METHOD TryMakeReferenceTo : BOOL
VAR_INPUT
	Target : I_Datatype;
END_VAR
VAR
	targetAsBit : I_BIT;
END_VAR
IF NOT Target.Root.TryResolveAs_BIT(targetAsBit) THEN
	RETURN;
END_IF

MakeReferenceTo(targetAsBit.Parent, targetAsBit.ByteOffset, targetAsBit.BitOffset);
TryMakeReferenceTo := TRUE;
END_METHOD

METHOD PUBLIC TryResolveAs_BIT : BOOL
VAR_INPUT
	Destination : REFERENCE TO I_BIT;
END_VAR
Destination := THIS^;
TryResolveAs_BIT := TRUE;
END_METHOD

PROPERTY PUBLIC TypeName : T_MAXSTRING
GET
TypeName := 'BIT';
END_GET
END_PROPERTY

PROPERTY PUBLIC Value : BOOL
GET
Value := GetBitValue();
END_GET
SET
SetBitValue(Value);
END_SET
END_PROPERTY

END_FUNCTION_BLOCK

// mobject-datatypes/Primitive/_NULL
{attribute 'linkalways'} 
{attribute 'no_explicit_call' := 'This FB is a CLASS and must be accessed using methods or properties'}
{attribute 'enable_dynamic_creation'}
FUNCTION_BLOCK _NULL EXTENDS DatatypeBase
VAR
END_VAR

PROPERTY PUBLIC Address : PVOID
GET
Address := 0;
END_GET
END_PROPERTY

METHOD PUBLIC ClearReference
VAR_INPUT
END_VAR
END_METHOD

METHOD PUBLIC Clone : I_Datatype
VAR
    pClone : POINTER TO _NULL;
END_VAR
pClone := __NEW(_NULL);
Clone := pClone^;
END_METHOD

PROPERTY PUBLIC IsNull : BOOL
GET
IsNull := TRUE;
END_GET
END_PROPERTY

METHOD PUBLIC SerializeWith
VAR_INPUT
	Serializer : I_Serializer;
END_VAR
Serializer.AddNull();
END_METHOD

PROPERTY PUBLIC Size : UDINT
GET
Size := 0;
END_GET
END_PROPERTY

METHOD TryDeserializeFrom : BOOL
VAR_INPUT
	Deserializer : I_Deserializer;
	Feedback : I_DeserializerFeedback;
END_VAR
END_METHOD

METHOD TryMakeReferenceTo : BOOL
VAR_INPUT
	Target : I_Datatype;
END_VAR
TryMakeReferenceTo := FALSE;
END_METHOD

PROPERTY PUBLIC TypeName : T_MAXSTRING
GET
TypeName := 'NULL';
END_GET
END_PROPERTY

END_FUNCTION_BLOCK

// mobject-datatypes/Primitive/_PVOID
{attribute 'linkalways'} 
{attribute 'no_explicit_call' := 'This FB is a CLASS and must be accessed using methods or properties'}
{attribute 'enable_dynamic_creation'}
FUNCTION_BLOCK _PVOID EXTENDS DatatypeBase IMPLEMENTS I_PVOID
VAR
	localData : PVOID;
	activeData : REFERENCE TO PVOID REF= localData;
END_VAR

PROPERTY PUBLIC Address : PVOID
GET
Address := ADR(activeData);
END_GET
END_PROPERTY

METHOD PUBLIC ClearReference
VAR_INPUT
END_VAR
activeData REF= localData;
END_METHOD

METHOD PUBLIC Clone : I_Datatype
VAR
    pClone : POINTER TO _PVOID;
END_VAR
pClone := __NEW(_PVOID);
Clone := pClone^;
END_METHOD

METHOD PUBLIC MakeReferenceTo
VAR_INPUT
	ReferenceTarget : REFERENCE TO PVOID;
END_VAR
activeData REF= ReferenceTarget;
END_METHOD

METHOD PUBLIC SerializeWith
VAR_INPUT
	Serializer : I_Serializer;
END_VAR
VAR
	pVoidAsString : T_MAXSTRING;
END_VAR
pVoidAsString := pvoid_To_string(activeData);
Serializer.AddString(pVoidAsString);
END_METHOD

PROPERTY PUBLIC Size : UDINT
GET
Size := SIZEOF(activeData);
END_GET
END_PROPERTY

METHOD TryDeserializeFrom : BOOL
VAR_INPUT
	Deserializer : I_Deserializer;
	Feedback : I_DeserializerFeedback;
END_VAR
VAR
	pVoidAsString : T_MAXSTRING;
END_VAR
IF NOT Deserializer.TryGetString(pVoidAsString, Feedback) THEN
	RETURN;
END_IF

activeData := STRING_TO_PVOID(pVoidAsString);
TryDeserializeFrom := TRUE;
END_METHOD

METHOD TryMakeReferenceTo : BOOL
VAR_INPUT
	Target : I_Datatype;
END_VAR
VAR
	pTargetData : POINTER TO PVOID;
END_VAR
IF NOT IsEquivalentTo(Target) THEN
	RETURN;
END_IF

pTargetData := Target.Address;
activeData REF= pTargetData^;
TryMakeReferenceTo := TRUE;
END_METHOD

METHOD PUBLIC TryResolveAs_PVOID : BOOL
VAR_INPUT
	Destination : REFERENCE TO I_PVOID;
END_VAR
Destination := THIS^;
TryResolveAs_PVOID := TRUE;
END_METHOD

PROPERTY PUBLIC TypeName : T_MAXSTRING
GET
TypeName := 'PVOID';
END_GET
END_PROPERTY

{warning disable C5410}
PROPERTY PUBLIC Value : REFERENCE TO PVOID
{warning restore C5410}
GET
Value REF= activeData;
END_GET
END_PROPERTY

END_FUNCTION_BLOCK

// mobject-datatypes/Primitive/_REFERENCE_TO
{attribute 'linkalways'} 
{attribute 'no_explicit_call' := 'This FB is a CLASS and must be accessed using methods or properties'}
{attribute 'enable_dynamic_creation'}
FUNCTION_BLOCK _REFERENCE_TO EXTENDS Disposable IMPLEMENTS I_REFERENCE_TO
VAR
	nullTarget : _NULL;
	_target : I_Datatype := nullTarget;
END_VAR

//FB_Init is always available implicitly and it is used primarily for initialization.
//The return value is not evaluated. For a specific influence, you can also declare the
//methods explicitly and provide additional code there with the standard initialization
//code. You can evaluate the return value.
METHOD FB_Init: BOOL
VAR_INPUT
    bInitRetains: BOOL; // TRUE: the retain variables are initialized (reset warm / reset cold)
    bInCopyCode: BOOL;  // TRUE: the instance will be copied to the copy code afterward (online change)  
	RefTo : I_Datatype; 
END_VAR
IF RefTo = 0 THEN
	RETURN;
END_IF

this^._target := RefTo;
END_METHOD

METHOD PUBLIC Accept
VAR_INPUT
	Visitor : I_DatatypeVisitor;
END_VAR
Visitor.VisitDatatype(THIS^);
END_METHOD

PROPERTY PUBLIC Address : PVOID
GET
Address := _target.Address;
END_GET
END_PROPERTY

METHOD PUBLIC ClearReference
VAR_INPUT
END_VAR
_target := nullTarget;
END_METHOD

METHOD PUBLIC Clone : I_Datatype
VAR
    pClone : POINTER TO _REFERENCE_TO;
END_VAR
pClone := __NEW(_REFERENCE_TO(RefTo := _target));
Clone := pClone^;
END_METHOD

METHOD PUBLIC IsEquivalentTo : BOOL
VAR_INPUT
	Datatype : I_Datatype;
END_VAR
IsEquivalentTo := _target.IsEquivalentTo(Datatype);
END_METHOD

PROPERTY PUBLIC IsNull : BOOL
GET
IsNull := _target.IsNull;
END_GET
END_PROPERTY

PROPERTY PUBLIC IsUserDefined : BOOL
GET
IsUserDefined := _target.IsUserDefined;
END_GET
END_PROPERTY

PROPERTY PUBLIC IsValidReference : BOOL
GET
IF _target.IsNull THEN
	RETURN;
END_IF

IsValidReference := TRUE;
END_GET
END_PROPERTY

PROPERTY PUBLIC Root : I_Datatype
GET
IF _target.IsNull THEN
	Root := THIS^;
	RETURN;
END_IF

Root := _target.Root;
END_GET
END_PROPERTY

METHOD PUBLIC SerializeTypeWith
VAR_INPUT
	Serializer : I_Serializer;
END_VAR
Serializer.StartObject();
Serializer.AddKeyString('typeName',TypeName);
Serializer.EndObject();
END_METHOD

METHOD PUBLIC SerializeWith
VAR_INPUT
	Serializer : I_Serializer;
END_VAR
_target.SerializeWith(Serializer);
END_METHOD

PROPERTY PUBLIC Size : UDINT
GET
Size := _target.Size;
END_GET
END_PROPERTY

METHOD PUBLIC TryConvertTo : BOOL
VAR_INPUT
	Destination : ANY;
END_VAR
TryConvertTo := _target.TryConvertTo(Destination);
END_METHOD

METHOD PUBLIC TryConvertTo_ : BOOL
VAR_INPUT
	Destination : I_Datatype;
END_VAR
TryConvertTo_ := _target.TryConvertTo_(Destination);
END_METHOD

METHOD PUBLIC TryCopyFrom : BOOL
VAR_INPUT
	Source : I_Datatype;
END_VAR
TryCopyFrom := _target.TryCopyFrom(Source);
END_METHOD

METHOD TryDeserializeFrom : BOOL
VAR_INPUT
	Deserializer : I_Deserializer;
	Feedback : I_DeserializerFeedback;
END_VAR
TryDeserializeFrom := _target.TryDeserializeFrom(Deserializer, Feedback);
END_METHOD

METHOD TryMakeReferenceTo : BOOL
VAR_INPUT
	Target : I_Datatype;
END_VAR
IF Target = 0 THEN
	RETURN;
END_IF

_target := Target;
TryMakeReferenceTo := TRUE;
END_METHOD

METHOD PUBLIC TryResolveAs_ANY : BOOL
VAR_INPUT
	Destination : REFERENCE TO I_ANY;
END_VAR
TryResolveAs_ANY := _target.TryResolveAs_ANY(Destination);
END_METHOD

METHOD PUBLIC TryResolveAs_BIT : BOOL
VAR_INPUT
	Destination : REFERENCE TO I_BIT;
END_VAR
TryResolveAs_BIT := _target.TryResolveAs_BIT(Destination);
END_METHOD

METHOD PUBLIC TryResolveAs_BOOL : BOOL
VAR_INPUT
	Destination : REFERENCE TO I_BOOL;
END_VAR
TryResolveAs_BOOL := _target.TryResolveAs_BOOL(Destination);
END_METHOD

METHOD PUBLIC TryResolveAs_BYTE : BOOL
VAR_INPUT
	Destination : REFERENCE TO I_BYTE;
END_VAR
TryResolveAs_BYTE := _target.TryResolveAs_BYTE(Destination);
END_METHOD

METHOD PUBLIC TryResolveAs_DINT : BOOL
VAR_INPUT
	Destination : REFERENCE TO I_DINT;
END_VAR
TryResolveAs_DINT := _target.TryResolveAs_DINT(Destination);
END_METHOD

METHOD PUBLIC TryResolveAs_DT : BOOL
VAR_INPUT
	Destination : REFERENCE TO I_DT;
END_VAR
TryResolveAs_DT := _target.TryResolveAs_DT(Destination);
END_METHOD

METHOD PUBLIC TryResolveAs_DWORD : BOOL
VAR_INPUT
	Destination : REFERENCE TO I_DWORD;
END_VAR
TryResolveAs_DWORD := _target.TryResolveAs_DWORD(Destination);
END_METHOD

METHOD PUBLIC TryResolveAs_INT : BOOL
VAR_INPUT
	Destination : REFERENCE TO I_INT;
END_VAR
TryResolveAs_INT := _target.TryResolveAs_INT(Destination);
END_METHOD

METHOD PUBLIC TryResolveAs_LINT : BOOL
VAR_INPUT
	Destination : REFERENCE TO I_LINT;
END_VAR
TryResolveAs_LINT := _target.TryResolveAs_LINT(Destination);
END_METHOD

METHOD PUBLIC TryResolveAs_LREAL : BOOL
VAR_INPUT
	Destination : REFERENCE TO I_LREAL;
END_VAR
TryResolveAs_LREAL := _target.TryResolveAs_LREAL(Destination);
END_METHOD

METHOD PUBLIC TryResolveAs_LWORD : BOOL
VAR_INPUT
	Destination : REFERENCE TO I_LWORD;
END_VAR
TryResolveAs_LWORD := _target.TryResolveAs_LWORD(Destination);
END_METHOD

METHOD PUBLIC TryResolveAs_PVOID : BOOL
VAR_INPUT
	Destination : REFERENCE TO I_PVOID;
END_VAR
TryResolveAs_PVOID := _target.TryResolveAs_PVOID(Destination);
END_METHOD

METHOD PUBLIC TryResolveAs_REAL : BOOL
VAR_INPUT
	Destination : REFERENCE TO I_REAL;
END_VAR
TryResolveAs_REAL := _target.TryResolveAs_REAL(Destination);
END_METHOD

METHOD PUBLIC TryResolveAs_REFERENCE_TO : BOOL
VAR_INPUT
	Destination : REFERENCE TO I_REFERENCE_TO;
END_VAR
Destination := THIS^;
TryResolveAs_REFERENCE_TO := TRUE;
END_METHOD

METHOD PUBLIC TryResolveAs_SINT : BOOL
VAR_INPUT
	Destination : REFERENCE TO I_SINT;
END_VAR
TryResolveAs_SINT := _target.TryResolveAs_SINT(Destination);
END_METHOD

METHOD PUBLIC TryResolveAs_STRING : BOOL
VAR_INPUT
	Destination : REFERENCE TO I_STRING;
END_VAR
TryResolveAs_STRING := _target.TryResolveAs_STRING(Destination);
END_METHOD

METHOD PUBLIC TryResolveAs_TIME_OF_DAY : BOOL
VAR_INPUT
	Destination : REFERENCE TO I_TIME_OF_DAY;
END_VAR
TryResolveAs_TIME_OF_DAY := _target.TryResolveAs_TIME_OF_DAY(Destination);
END_METHOD

METHOD PUBLIC TryResolveAs_TOD : BOOL
VAR_INPUT
	Destination : REFERENCE TO I_TOD;
END_VAR
TryResolveAs_TOD := _target.TryResolveAs_TOD(Destination);
END_METHOD

METHOD PUBLIC TryResolveAs_UDINT : BOOL
VAR_INPUT
	Destination : REFERENCE TO I_UDINT;
END_VAR
TryResolveAs_UDINT := _target.TryResolveAs_UDINT(Destination);
END_METHOD

METHOD PUBLIC TryResolveAs_UINT : BOOL
VAR_INPUT
	Destination : REFERENCE TO I_UINT;
END_VAR
TryResolveAs_UINT := _target.TryResolveAs_UINT(Destination);
END_METHOD

METHOD PUBLIC TryResolveAs_ULINT : BOOL
VAR_INPUT
	Destination : REFERENCE TO I_ULINT;
END_VAR
TryResolveAs_ULINT := _target.TryResolveAs_ULINT(Destination);
END_METHOD

METHOD PUBLIC TryResolveAs_USINT : BOOL
VAR_INPUT
	Destination : REFERENCE TO I_USINT;
END_VAR
TryResolveAs_USINT := _target.TryResolveAs_USINT(Destination);
END_METHOD

METHOD PUBLIC TryResolveAs_WORD : BOOL
VAR_INPUT
	Destination : REFERENCE TO I_WORD;
END_VAR
TryResolveAs_WORD := _target.TryResolveAs_WORD(Destination);
END_METHOD

METHOD PUBLIC TryResolveAsAliasDatatype : BOOL
VAR_INPUT
	Destination : REFERENCE TO I_AliasDatatype;
END_VAR
TryResolveAsAliasDatatype := _target.TryResolveAsAliasDatatype(Destination);
END_METHOD

METHOD PUBLIC TryResolveAsArrayDatatype : BOOL
VAR_INPUT
	Destination : REFERENCE TO I_ArrayDatatype;
END_VAR
TryResolveAsArrayDatatype := _target.TryResolveAsArrayDatatype(Destination);
END_METHOD

METHOD PUBLIC TryResolveAsBitDatatype : BOOL
VAR_INPUT
	Destination : REFERENCE TO I_BIT;
END_VAR
TryResolveAsBitDatatype := _target.TryResolveAsBitDatatype(Destination);
END_METHOD

METHOD PUBLIC TryResolveAsEnumDatatype : BOOL
VAR_INPUT
	Destination : REFERENCE TO I_EnumDatatype;
END_VAR
TryResolveAsEnumDatatype := _target.TryResolveAsEnumDatatype(Destination);
END_METHOD

METHOD PUBLIC TryResolveAsInterfaceDatatype : BOOL
VAR_INPUT
	Destination : REFERENCE TO I_InterfaceDatatype;
END_VAR
TryResolveAsInterfaceDatatype := _target.TryResolveAsInterfaceDatatype(Destination);
END_METHOD

METHOD PUBLIC TryResolveAsStructuredDatatype : BOOL
VAR_INPUT
	Destination : REFERENCE TO I_StructuredDatatype;
END_VAR
TryResolveAsStructuredDatatype := _target.TryResolveAsStructuredDatatype(Destination);
END_METHOD

METHOD PUBLIC TryResolveAsUserDefinedDatatype : BOOL
VAR_INPUT
	Destination : REFERENCE TO I_UserDefinedDatatype;
END_VAR
TryResolveAsUserDefinedDatatype := _target.TryResolveAsUserDefinedDatatype(Destination);
END_METHOD

PROPERTY PUBLIC TypeName : T_MAXSTRING
GET
TypeName := concat('REFERENCE TO ', _target.TypeName);
END_GET
END_PROPERTY

END_FUNCTION_BLOCK

// mobject-datatypes/Primitive/_TIME_OF_DAY
{attribute 'linkalways'} 
{attribute 'no_explicit_call' := 'This FB is a CLASS and must be accessed using methods or properties'}
{attribute 'enable_dynamic_creation'}
FUNCTION_BLOCK _TIME_OF_DAY EXTENDS DatatypeBase IMPLEMENTS I_TIME_OF_DAY
VAR
	localData : TIME_OF_DAY;
	activeData : REFERENCE TO TIME_OF_DAY REF= localData;
END_VAR

METHOD FB_init : BOOL
VAR_INPUT
	bInitRetains : BOOL; // if TRUE, the retain variables are initialized (warm start / cold start)
	bInCopyCode : BOOL;  // if TRUE, the instance afterwards gets moved WORDo the copy code (online change)
	InitialValue : TIME_OF_DAY;
END_VAR
localData := InitialValue;
END_METHOD

PROPERTY PUBLIC Address : PVOID
GET
Address := ADR(activeData);
END_GET
END_PROPERTY

METHOD PUBLIC ClearReference
VAR_INPUT
END_VAR
activeData REF= localData;
END_METHOD

METHOD PUBLIC Clone : I_Datatype
VAR
    pClone : POINTER TO _TIME_OF_DAY;
END_VAR
pClone := __NEW(_TIME_OF_DAY(InitialValue := Value));
Clone := pClone^;
END_METHOD

METHOD PUBLIC MakeReferenceTo
VAR_INPUT
	ReferenceTarget : REFERENCE TO TIME_OF_DAY;
END_VAR
activeData REF= ReferenceTarget;
END_METHOD

METHOD PUBLIC SerializeWith
VAR_INPUT
	Serializer : I_Serializer;
END_VAR
Serializer.AddTod(activeData);
END_METHOD

PROPERTY PUBLIC Size : UDINT
GET
Size := SIZEOF(activeData);
END_GET
END_PROPERTY

METHOD TryDeserializeFrom : BOOL
VAR_INPUT
	Deserializer : I_Deserializer;
	Feedback : I_DeserializerFeedback;
END_VAR
TryDeserializeFrom := Deserializer.TryGetTod(activeData, Feedback);
END_METHOD

METHOD TryMakeReferenceTo : BOOL
VAR_INPUT
	Target : I_Datatype;
END_VAR
VAR
	pTargetData : POINTER TO TIME_OF_DAY;
END_VAR
IF NOT IsEquivalentTo(Target) THEN
	RETURN;
END_IF

pTargetData := Target.Address;
activeData REF= pTargetData^;
TryMakeReferenceTo := TRUE;
END_METHOD

METHOD PUBLIC TryResolveAs_TIME_OF_DAY : BOOL
VAR_INPUT
	Destination : REFERENCE TO I_TIME_OF_DAY;
END_VAR
Destination := THIS^;
TryResolveAs_TIME_OF_DAY := TRUE;
END_METHOD

PROPERTY PUBLIC TypeName : T_MAXSTRING
GET
TypeName := 'TIME_OF_DAY';
END_GET
END_PROPERTY

{warning disable C5410}
PROPERTY PUBLIC Value : REFERENCE TO TIME_OF_DAY
{warning restore C5410}
GET
Value REF= activeData;
END_GET
END_PROPERTY

END_FUNCTION_BLOCK

// mobject-deserialization/DeserializationFeedback/DeserializerFeedback
{attribute 'linkalways'} 
{attribute 'no_explicit_call' := 'This FB is a CLASS and must be accessed using methods or properties'}
{attribute 'enable_dynamic_creation'}
FUNCTION_BLOCK DeserializerFeedback IMPLEMENTS I_DeserializerFeedback
VAR
	errors : Stack;
	_hasError : BOOL;
	nullError : NullError;
	deserializationErrorFactory : DeserializationErrorFactory;
END_VAR

METHOD FB_exit : BOOL
VAR_INPUT
	bInCopyCode : BOOL; // if TRUE, the exit method is called for exiting an instance that is copied afterwards (online change).
END_VAR
IF bInCopyCode THEN
	RETURN;
END_IF

DisposeErrors();
END_METHOD

METHOD PRIVATE DisposeErrors : BOOL
VAR
	error : I_Error;
END_VAR
WHILE errors.TryPop(error) DO
	error.Dispose();
END_WHILE
END_METHOD

PROPERTY PUBLIC FirstError : I_Error
GET
VAR
	error : I_Error;
END_VAR
IF NOT HasError THEN
	FirstError := nullError;
	RETURN;
END_IF

IF NOT errors.TryPeek(error) THEN
	FirstError := nullError;
	RETURN;
END_IF

FirstError := error;
END_GET
END_PROPERTY

PROPERTY PUBLIC HasError : BOOL
GET
HasError := _hasError;
END_GET
END_PROPERTY

METHOD PUBLIC LogDeserializationFailedError
VAR_INPUT
	Message : T_MAXSTRING;
END_VAR
LogError(deserializationErrorFactory.CreateCustomDeserializationFailedError(Message));
END_METHOD

METHOD PUBLIC LogError
VAR_INPUT
	Error : I_Error;
END_VAR
errors.Push(Error);
_hasError := TRUE;
END_METHOD

METHOD PUBLIC LogIncorrectKeyTypeError
VAR_INPUT
	ExpectedType : T_MAXSTRING;
	ActualKey : T_MAXSTRING;
END_VAR
LogError(deserializationErrorFactory.CreateIncorrectKeyTypeError(ExpectedType, ActualKey));
END_METHOD

METHOD PUBLIC LogIncorrectTypeError
VAR_INPUT
	ExpectedType : T_MAXSTRING;
END_VAR
LogError(deserializationErrorFactory.CreateIncorrectTypeError(ExpectedType));
END_METHOD

METHOD PUBLIC LogInvalidKeyError
VAR_INPUT
END_VAR
LogError(deserializationErrorFactory.CreateInvalidKeyError());
END_METHOD

METHOD PUBLIC LogMissingKeyError
VAR_INPUT
	ExpectedKey : T_MAXSTRING;
END_VAR
LogError(deserializationErrorFactory.CreateMissingKeyError(ExpectedKey));
END_METHOD

METHOD PUBLIC Reset : BOOL
VAR_INPUT
END_VAR
DisposeErrors();
_hasError := FALSE;
END_METHOD

METHOD PUBLIC SerializeWith
VAR_INPUT
	Serializer : I_Serializer;
END_VAR
VAR
	enumerator : I_ForwardEnumerator;
	error : I_Error;
END_VAR
IF NOT HasError THEN
	RETURN;
END_IF

Serializer.AddKey('errors');
Serializer.StartArray();

enumerator := errors.GetEnumerator();

WHILE enumerator.MoveNext() DO
	IF enumerator.TryGet(error) THEN
		error.SerializeWith(Serializer);
	END_IF
END_WHILE

enumerator.Dispose();
Serializer.EndArray();
END_METHOD

END_FUNCTION_BLOCK

// mobject-errors/Errors/NullError
{attribute 'linkalways'} 
{attribute 'no_explicit_call' := 'This FB is a CLASS and must be accessed using methods or properties'}
{attribute 'enable_dynamic_creation'}
FUNCTION_BLOCK NullError EXTENDS Error
VAR
END_VAR

PROPERTY ErrorType : T_MAXSTRING
GET
END_GET
END_PROPERTY

PROPERTY PUBLIC Message : T_MAXSTRING
GET
END_GET
END_PROPERTY

METHOD PUBLIC SerializeWith
VAR_INPUT
	Serializer : I_Serializer;
END_VAR
END_METHOD

END_FUNCTION_BLOCK

// mobject-deserialization/Errors/DeserializationErrorFactory
{attribute 'linkalways'} 
{attribute 'no_explicit_call' := 'This FB is a CLASS and must be accessed using methods or properties'}
{attribute 'enable_dynamic_creation'}
FUNCTION_BLOCK DeserializationErrorFactory
VAR
END_VAR

METHOD PUBLIC CreateCustomDeserializationFailedError : I_Error
VAR_INPUT
	CustomMessage : T_MAXSTRING;
END_VAR
VAR
	pError : POINTER TO CustomDeserializationFailedError;
END_VAR
pError := __NEW(CustomDeserializationFailedError(Message := CustomMessage));
CreateCustomDeserializationFailedError := pError^;
END_METHOD

METHOD PUBLIC CreateIncorrectKeyTypeError : I_Error
VAR_INPUT
	ExpectedType : T_MAXSTRING;
	ActualKey : T_MAXSTRING;
END_VAR
VAR
	pError : POINTER TO IncorrectKeyTypeDeserializationError;
END_VAR
pError := __NEW(IncorrectKeyTypeDeserializationError(DataType := ExpectedType, Key := ActualKey));
CreateIncorrectKeyTypeError := pError^;
END_METHOD

METHOD PUBLIC CreateIncorrectTypeError : I_Error
VAR_INPUT
	ExpectedType : T_MAXSTRING;
END_VAR
VAR
	pError : POINTER TO IncorrectTypeDeserializationError;
END_VAR
pError := __NEW(IncorrectTypeDeserializationError(DataType := ExpectedType));
CreateIncorrectTypeError := pError^;
END_METHOD

METHOD PUBLIC CreateInvalidArrayIndexError : I_Error
VAR_INPUT
	AttemptedIndex : UDINT;
END_VAR
VAR
	pError : POINTER TO InvalidArrayIndexDeserializationError;
END_VAR
pError := __NEW(InvalidArrayIndexDeserializationError(Index := AttemptedIndex));
CreateInvalidArrayIndexError := pError^;
END_METHOD

METHOD PUBLIC CreateInvalidKeyError : I_Error
VAR_INPUT
END_VAR
VAR
	pError : POINTER TO InvalidKeyDeserializationError;
END_VAR
pError := __NEW(InvalidKeyDeserializationError);
CreateInvalidKeyError := pError^;
END_METHOD

METHOD PUBLIC CreateMissingKeyError : I_Error
VAR_INPUT
	ExpectedKey : T_MAXSTRING;
END_VAR
VAR
	pError : POINTER TO MissingKeyDeserializationError;
END_VAR
pError := __NEW(MissingKeyDeserializationError(Key := ExpectedKey));
CreateMissingKeyError := pError^;
END_METHOD

END_FUNCTION_BLOCK

// mobject-deserialization/Errors/CustomError/CustomDeserializationFailedError
{attribute 'linkalways'} 
{attribute 'no_explicit_call' := 'This FB is a CLASS and must be accessed using methods or properties'}
{attribute 'enable_dynamic_creation'}
FUNCTION_BLOCK CustomDeserializationFailedError EXTENDS Error
VAR
	_message : T_MAXSTRING;
END_VAR

METHOD FB_init : BOOL
VAR_INPUT
	bInitRetains : BOOL; // if TRUE, the retain variables are initialized (warm start / cold start)
	bInCopyCode : BOOL;  // if TRUE, the instance afterwards gets moved into the copy code (online change)
	Message : T_MAXSTRING;
END_VAR
this^._message := Message;
END_METHOD

PROPERTY PUBLIC ErrorType : T_MAXSTRING
GET
ErrorType := 'CUSTOM_DESERIALIZATION_ERROR';
END_GET
END_PROPERTY

PROPERTY PUBLIC Message : T_MAXSTRING
GET
Message := CONCAT('Deserialization Failed, ',_message);
END_GET
END_PROPERTY

END_FUNCTION_BLOCK

// mobject-deserialization/Errors/IncorrectType/IncorrectKeyTypeDeserializationError
{attribute 'linkalways'} 
{attribute 'no_explicit_call' := 'This FB is a CLASS and must be accessed using methods or properties'}
{attribute 'enable_dynamic_creation'}
FUNCTION_BLOCK IncorrectKeyTypeDeserializationError EXTENDS IncorrectTypeDeserializationError
VAR
	key : T_MAXSTRING;
END_VAR

METHOD FB_init : BOOL
VAR_INPUT
	bInitRetains : BOOL; // if TRUE, the retain variables are initialized (warm start / cold start)
	bInCopyCode : BOOL;  // if TRUE, the instance afterwards gets moved into the copy code (online change)
	DataType : T_MAXSTRING;
	Key : T_MAXSTRING;
END_VAR
THIS^.key := Key;
END_METHOD

PROPERTY PUBLIC Message : T_MAXSTRING
GET
VAR
	messageWithKey : T_MAXSTRING;
END_VAR
messageWithKey := concat(' for key : ',key);
Message := CONCAT(SUPER^.Message, messageWithKey);
END_GET
END_PROPERTY

END_FUNCTION_BLOCK

// mobject-deserialization/Errors/IncorrectType/IncorrectTypeDeserializationError
{attribute 'linkalways'} 
{attribute 'no_explicit_call' := 'This FB is a CLASS and must be accessed using methods or properties'}
{attribute 'enable_dynamic_creation'}
FUNCTION_BLOCK IncorrectTypeDeserializationError EXTENDS Error
VAR
	dataType : T_MAXSTRING;
END_VAR

METHOD FB_init : BOOL
VAR_INPUT
	bInitRetains : BOOL; // if TRUE, the retain variables are initialized (warm start / cold start)
	bInCopyCode : BOOL;  // if TRUE, the instance afterwards gets moved into the copy code (online change)
	DataType : T_MAXSTRING;
END_VAR
THIS^.dataType := DataType;
END_METHOD

PROPERTY PUBLIC ErrorType : T_MAXSTRING
GET
ErrorType := 'INCORRECT_DATATYPE_DESERIALIZATION_ERROR';
END_GET
END_PROPERTY

PROPERTY PUBLIC Message : T_MAXSTRING
GET
Message := CONCAT('Deserialization Failed, Incorrect Datatype : ', dataType);
END_GET
END_PROPERTY

END_FUNCTION_BLOCK

// mobject-deserialization/Errors/Invalid Index/InvalidArrayIndexDeserializationError
{attribute 'linkalways'} 
{attribute 'no_explicit_call' := 'This FB is a CLASS and must be accessed using methods or properties'}
{attribute 'enable_dynamic_creation'}
FUNCTION_BLOCK InvalidArrayIndexDeserializationError EXTENDS Error
VAR
	index : UDINT;
END_VAR

METHOD FB_init : BOOL
VAR_INPUT
	bInitRetains : BOOL; // if TRUE, the retain variables are initialized (warm start / cold start)
	bInCopyCode : BOOL;  // if TRUE, the instance afterwards gets moved into the copy code (online change)
	Index : UDINT;
END_VAR
this^.index := Index;
END_METHOD

PROPERTY PUBLIC ErrorType : T_MAXSTRING
GET
ErrorType := 'INVALID_ARRAY_INDEX_DESERIALIZATION_ERROR';
END_GET
END_PROPERTY

PROPERTY PUBLIC Message : T_MAXSTRING
GET
Message := CONCAT('Deserialization Failed, Array Index Out Of Bounds ', UDINT_TO_STRING(index));
END_GET
END_PROPERTY

END_FUNCTION_BLOCK

// mobject-deserialization/Errors/Invalid Key/InvalidKeyDeserializationError
{attribute 'linkalways'} 
{attribute 'no_explicit_call' := 'This FB is a CLASS and must be accessed using methods or properties'}
{attribute 'enable_dynamic_creation'}
FUNCTION_BLOCK InvalidKeyDeserializationError EXTENDS Error
VAR
END_VAR

PROPERTY PUBLIC ErrorType : T_MAXSTRING
GET
ErrorType := 'INVALID_KEY_DESERIALIZATION_ERROR';
END_GET
END_PROPERTY

PROPERTY PUBLIC Message : T_MAXSTRING
GET
Message := 'Deserialization Failed, Key Cannot Be Empty';
END_GET
END_PROPERTY

END_FUNCTION_BLOCK

// mobject-deserialization/Errors/Missing Key/MissingKeyDeserializationError
{attribute 'linkalways'} 
{attribute 'no_explicit_call' := 'This FB is a CLASS and must be accessed using methods or properties'}
{attribute 'enable_dynamic_creation'}
FUNCTION_BLOCK MissingKeyDeserializationError EXTENDS Error
VAR
	key : T_MAXSTRING;
END_VAR

METHOD FB_init : BOOL
VAR_INPUT
	bInitRetains : BOOL; // if TRUE, the retain variables are initialized (warm start / cold start)
	bInCopyCode : BOOL;  // if TRUE, the instance afterwards gets moved into the copy code (online change)
	Key : T_MAXSTRING;
END_VAR
this^.key := Key;
END_METHOD

PROPERTY PUBLIC ErrorType : T_MAXSTRING
GET
ErrorType := 'MISSING_KEY_DESERIALIZATION_ERROR';
END_GET
END_PROPERTY

PROPERTY PUBLIC Message : T_MAXSTRING
GET
Message := CONCAT('Deserialization Failed, Missing Key : ',key);
END_GET
END_PROPERTY

END_FUNCTION_BLOCK

// mobject-deserialization/GarbageCollector/DeserializerGarbageCollector
{attribute 'linkalways'} 
{attribute 'no_explicit_call' := 'This FB is a CLASS and must be accessed using methods or properties'}
{attribute 'enable_dynamic_creation'}
FUNCTION_BLOCK DeserializerGarbageCollector EXTENDS Disposable Implements I_DeserializerGarbageCollector
VAR
	deserializers : Stack;
END_VAR

METHOD FB_exit : BOOL
VAR_INPUT
	bInCopyCode : BOOL; // if TRUE, the exit method is called for exiting an instance that is copied afterwards (online change).
END_VAR
IF bInCopyCode THEN
	RETURN;
END_IF

DisposeAll();
END_METHOD

METHOD PROTECTED DisposeAll
VAR
	deserializer : I_Deserializer;
END_VAR
WHILE deserializers.TryPop(deserializer) DO
	deserializer.Dispose();
END_WHILE
END_METHOD

METHOD PUBLIC Deregister
VAR_INPUT
	Deserializer : I_Deserializer;
END_VAR
deserializers.TryRemoveItem(Deserializer);
END_METHOD

METHOD PUBLIC Execute
VAR_INPUT
END_VAR
DisposeAll();
END_METHOD

METHOD PUBLIC Register
VAR_INPUT
	Deserializer : I_Deserializer;
END_VAR
deserializers.Push(Deserializer);
END_METHOD

END_FUNCTION_BLOCK

// mobject-deserialization/GarbageCollector/I_DeserializerGarbageCollector
INTERFACE I_DeserializerGarbageCollector EXTENDS __SYSTEM.IQueryInterface

METHOD PUBLIC Deregister
VAR_INPUT
	Deserializer : I_Deserializer;
END_VAR
END_METHOD

METHOD PUBLIC Register
VAR_INPUT
	Deserializer : I_Deserializer;
END_VAR
END_METHOD

END_INTERFACE

// mobject-json/_Internal/Events/JsonDeserializerChangedEvent
{attribute 'linkalways'} 
{attribute 'no_explicit_call' := 'This FB is a CLASS and must be accessed using methods or properties'}
{attribute 'enable_dynamic_creation'}
FUNCTION_BLOCK JsonDeserializerChangedEvent EXTENDS JsonDeserializerEvent IMPLEMENTS I_JsonDeserializerChangedEvent

END_FUNCTION_BLOCK

// mobject-json/_Internal/Events/JsonDeserializerEvent
{attribute 'linkalways'} 
{attribute 'no_explicit_call' := 'This FB is a CLASS and must be accessed using methods or properties'}
{attribute 'enable_dynamic_creation'}
FUNCTION_BLOCK ABSTRACT JsonDeserializerEvent EXTENDS Disposable
VAR
	_target : I_JsonDeserializer;
END_VAR

METHOD FB_init : BOOL
VAR_INPUT
	bInitRetains : BOOL; // if TRUE, the retain variables are initialized (warm start / cold start)
	bInCopyCode : BOOL;  // if TRUE, the instance afterwards gets moved into the copy code (online change)
	Target : I_JsonDeserializer;
END_VAR
This^._target := Target;
END_METHOD

PROPERTY PUBLIC Target : I_JsonDeserializer
GET
PUBLIC
Target := _target;
END_GET
END_PROPERTY

END_FUNCTION_BLOCK

// mobject-json/JsonDeserializer/I_JsonDeserializer
INTERFACE I_JsonDeserializer EXTENDS I_Deserializer, I_EventEmitter, I_Disposable

END_INTERFACE

// mobject-json/JsonDeserializer/Events/I_JsonDeserializerChangedEvent
INTERFACE I_JsonDeserializerChangedEvent EXTENDS I_Event

PROPERTY PUBLIC Target : I_JsonDeserializer
GET
END_GET
END_PROPERTY

END_INTERFACE

// mobject-json/_Internal/Events/JsonDeserializerDisposedEvent
{attribute 'linkalways'} 
{attribute 'no_explicit_call' := 'This FB is a CLASS and must be accessed using methods or properties'}
{attribute 'enable_dynamic_creation'}
FUNCTION_BLOCK JsonDeserializerDisposedEvent EXTENDS JsonDeserializerEvent IMPLEMENTS I_JsonDeserializerDisposedEvent

END_FUNCTION_BLOCK

// mobject-json/JsonDeserializer/Events/I_JsonDeserializerDisposedEvent
INTERFACE I_JsonDeserializerDisposedEvent EXTENDS I_Event

PROPERTY PUBLIC Target : I_JsonDeserializer
GET
END_GET
END_PROPERTY

END_INTERFACE

// mobject-json/_Internal/JsonDeserializerForwardEnumerator/JsonDeserializerArrayForwardEnumerator
{attribute 'linkalways'} 
{attribute 'no_explicit_call' := 'This FB is a CLASS and must be accessed using methods or properties'}
{attribute 'enable_dynamic_creation'}
FUNCTION_BLOCK JsonDeserializerArrayForwardEnumerator EXTENDS Disposable IMPLEMENTS I_DeserializerArrayForwardEnumerator, I_EventHandler
VAR
	parent : I_JsonDeserializer;
	jsonParser : REFERENCE TO JsonDomParser;
	root : SJsonValue;
	garbageCollector : I_DeserializerGarbageCollector;
	nullNode : I_Deserializer;
	moveNextCalled : BOOL := FALSE;
	invalid : BOOL := FALSE; 
	nextArrayPosition : SJsonValue;
	arrayBeginPosition : SJsonValue;
	arrayEndPosition : SJsonValue;
	currentDeserializer : I_Deserializer;
	_index : DINT;
END_VAR

METHOD FB_init : BOOL
VAR_INPUT
	bInitRetains : BOOL; // if TRUE, the retain variables are initialized (warm start / cold start)
	bInCopyCode : BOOL;  // if TRUE, the instance afterwards gets moved into the copy code (online change)
	ParentJsonDeserializer : I_JsonDeserializer;
	ParentJsonDomParser : REFERENCE TO JsonDomParser;
	NodeRoot : SJsonValue;
	ParentGarbageCollector : I_DeserializerGarbageCollector;
	ParentNullDeserializer : I_Deserializer;
END_VAR
THIS^.parent := ParentJsonDeserializer;
THIS^.jsonParser REF= ParentJsonDomParser;
THIS^.root := NodeRoot;
THIS^.garbageCollector := ParentGarbageCollector;
THIS^.nullNode := ParentNullDeserializer;

Initialize();

Parent.OnEvent('OnChanged',THIS^);
Parent.OnEvent('OnDisposed',THIS^);
END_METHOD

METHOD FB_exit : BOOL
VAR_INPUT
	bInCopyCode : BOOL; // if TRUE, the exit method is called for exiting an instance that is copied afterwards (online change).
END_VAR
IF bInCopyCode THEN
	RETURN;
END_IF

IF parent = 0 THEN
	RETURN;
END_IF

parent.OffEvent('OnChanged',THIS^);
parent.OffEvent('OnDisposed',THIS^);
END_METHOD

METHOD PROTECTED CreateDeserializer : I_Deserializer
VAR_INPUT
	DeserializerRoot : SJsonValue;
END_VAR
VAR 
	pNode : POINTER TO JsonDeserializerNode;
END_VAR
pNode := __NEW(JsonDeserializerNode(
	ParentJsonDeserializer := parent,
	ParentJsonDomParser := jsonParser, 
	NodeRoot := DeserializerRoot, 
	ParentGarbageCollector := garbageCollector, 
	ParentNullDeserializer := nullNode
));

CreateDeserializer := pNode^;
END_METHOD

METHOD PROTECTED Initialize
VAR_INPUT
END_VAR
IF NOT jsonParser.IsArray(root) THEN
	invalid := TRUE;
	RETURN;
END_IF

arrayBeginPosition := jsonParser.ArrayBegin(root);
arrayEndPosition := jsonParser.ArrayEnd(root);

IF arrayBeginPosition = 0 THEN
	invalid := TRUE;
	RETURN;
END_IF

IF arrayEndPosition = 0 THEN
	invalid := TRUE;
	RETURN;
END_IF
END_METHOD

METHOD PROTECTED UpdateCurrentDeserializer
VAR_INPUT
	Root : SJsonValue;
END_VAR
VAR
	newRoot : SJsonValue;
END_VAR
IF currentDeserializer <> 0 THEN
	currentDeserializer.Dispose();
	currentDeserializer := 0;
END_IF

IF invalid THEN
	RETURN;
END_IF

newRoot := jsonParser.GetArrayValue(Root);

IF newRoot = 0 THEN
	RETURN;
END_IF

currentDeserializer := CreateDeserializer(newRoot);
END_METHOD

PROPERTY PUBLIC Current : I_Deserializer
GET
IF NOT IsValid THEN
	Current := nullNode;
	RETURN;
END_IF

IF currentDeserializer = 0 THEN
	Current := nullNode;
	RETURN;
END_IF

Current := currentDeserializer;
END_GET
END_PROPERTY

METHOD PUBLIC HandleEvent
VAR_INPUT
	Event : I_Event;
END_VAR
VAR
	changedEvent : I_JsonDeserializerChangedEvent;
	disposedEvent : I_JsonDeserializerDisposedEvent;
END_VAR
IF __QUERYINTERFACE(Event, changedEvent) THEN
	invalid := TRUE;
ELSIF __QUERYINTERFACE(Event, disposedEvent) THEN
	parent := 0;
	Dispose();
END_IF
END_METHOD

PROPERTY Index : DINT
GET
Index := _index;
END_GET
END_PROPERTY

PROPERTY PUBLIC IsValid : BOOL
GET
PUBLIC
IF invalid THEN
	RETURN;
END_IF

IF parent = 0 THEN
	RETURN;
END_IF

IsValid := TRUE;
END_GET
END_PROPERTY

METHOD PUBLIC MoveNext : BOOL
IF invalid THEN
    RETURN;
END_IF

// Handle the initial move
IF NOT moveNextCalled THEN
    moveNextCalled := TRUE;
    UpdateCurrentDeserializer(arrayBeginPosition);
	nextArrayPosition := jsonParser.NextArray(arrayBeginPosition);
	_index := _index + 1;
	MoveNext := TRUE;
    RETURN;
END_IF

// Handle subsequent moves
IF nextArrayPosition <> arrayEndPosition THEN
	UpdateCurrentDeserializer(nextArrayPosition);
	nextArrayPosition := jsonParser.NextArray(nextArrayPosition);
	_index := _index + 1;
	MoveNext := TRUE;
END_IF
END_METHOD

END_FUNCTION_BLOCK

// mobject-json/JsonDomParser/JsonDomParser
{attribute 'linkalways'} 
{attribute 'no_explicit_call' := 'This FB is a CLASS and must be accessed using methods or properties'}
{attribute 'enable_dynamic_creation'}
FUNCTION_BLOCK JsonDomParser EXTENDS FB_JsonDynDomParser
VAR
	currentlyParsingType : (NOTHING, DOT_NOTATION_PROPERTY, BRACKET_NOTATION_PROPERTY_OR_ARRAY, BRACKET_NOTATION_PROPERTY_ELEMENT, BRACKET_NOTATION_ARRAY_ELEMENT);
	readWriteDataType : FB_JsonReadWriteDataType;
END_VAR

METHOD PRIVATE TrySetBool : BOOL
VAR_INPUT
	JsonValue : SJsonValue;
	Source : ANY;
END_VAR
VAR
	_BOOL : BOOL;
END_VAR
IF Source.TypeClass <> __SYSTEM.TYPE_CLASS.TYPE_BOOL THEN	
	RETURN;
END_IF

memcpy(ADR(_BOOL),Source.pValue,DINT_TO_UDINT(Source.diSize));
SetBool(jsonValue,_BOOL);
TrySetBool := TRUE;
END_METHOD

METHOD PRIVATE TrySetDouble : BOOL
VAR_INPUT
	JsonValue : SJsonValue;
	Source : ANY;
END_VAR
VAR
	convertSuccessful : BOOL;
	_REAL : REAL;
	_LREAL : LREAL;
END_VAR
CASE Source.TypeClass OF 

	__SYSTEM.TYPE_CLASS.TYPE_REAL : 
		memcpy(ADR(_REAL),Source.pValue,DINT_TO_UDINT(Source.diSize));
		convertSuccessful := TryConvert_Source_TO_Destination(_REAL,_LREAL);
	
	__SYSTEM.TYPE_CLASS.TYPE_LREAL : 
		memcpy(ADR(_LREAL),Source.pValue,DINT_TO_UDINT(Source.diSize));
		convertSuccessful := TRUE;
		
ELSE 
		
	RETURN;
		
END_CASE

IF NOT convertSuccessful THEN
	RETURN;
END_IF

SetDouble(jsonValue,_LREAL);
TrySetDouble := TRUE;
END_METHOD

METHOD PRIVATE TrySetInt : BOOL
VAR_INPUT
	JsonValue : SJsonValue;
	Source : ANY;
END_VAR
VAR
	convertSuccessful : BOOL;
	_SINT : USINT;	
	_INT : UINT;
	_DINT : DINT;
END_VAR
CASE Source.TypeClass OF
		
	__SYSTEM.TYPE_CLASS.TYPE_SINT : 
		memcpy(ADR(_SINT),Source.pValue,DINT_TO_UDINT(Source.diSize));
		convertSuccessful := TryConvert_Source_TO_Destination(_SINT,_DINT);
		
	__SYSTEM.TYPE_CLASS.TYPE_INT : 
		memcpy(ADR(_INT),Source.pValue,DINT_TO_UDINT(Source.diSize));
		convertSuccessful := TryConvert_Source_TO_Destination(_INT,_DINT);
		
	__SYSTEM.TYPE_CLASS.TYPE_DINT : 
		memcpy(ADR(_DINT),Source.pValue,DINT_TO_UDINT(Source.diSize));
		convertSuccessful := TRUE;
		
ELSE 
		
	RETURN;
		
END_CASE

IF NOT convertSuccessful THEN
	RETURN;
END_IF

SetInt(jsonValue,_DINT); // Not a typo, SetInt actually takes a DINT
TrySetInt := TRUE;
END_METHOD

METHOD PRIVATE TrySetInt64 : BOOL
VAR_INPUT
	JsonValue : SJsonValue;
	Source : ANY;
END_VAR
VAR
	_LINT : LINT;
END_VAR
IF Source.TypeClass <> __SYSTEM.TYPE_CLASS.TYPE_LINT THEN	
	RETURN;
END_IF

memcpy(ADR(_LINT),Source.pValue,DINT_TO_UDINT(Source.diSize));
SetInt64(jsonValue,_LINT);
TrySetInt64 := TRUE;
END_METHOD

METHOD PRIVATE TrySetString : BOOL
VAR_INPUT
	JsonValue : SJsonValue;
	Source : ANY;
END_VAR
VAR
	_STRING : POINTER TO STRING(1);
END_VAR
IF Source.TypeClass <> __SYSTEM.TYPE_CLASS.TYPE_STRING THEN	
	RETURN;
END_IF

_STRING := Source.pValue;

SetString(jsonValue,_STRING^);
TrySetString := TRUE;
END_METHOD

METHOD PRIVATE TrySetUint : BOOL
VAR_INPUT
	JsonValue : SJsonValue;
	Source : ANY;
END_VAR
VAR
	convertSuccessful : BOOL;
	_BYTE : BYTE;
	_WORD : WORD;
	_DWORD : DWORD;	
	_USINT : USINT;	
	_UINT : UINT;
	_UDINT : UDINT;
END_VAR
CASE Source.TypeClass OF 

	__SYSTEM.TYPE_CLASS.TYPE_BYTE : 
		memcpy(ADR(_BYTE),Source.pValue,DINT_TO_UDINT(Source.diSize));
		convertSuccessful := TryConvert_Source_TO_Destination(_BYTE,_UDINT);
	
	__SYSTEM.TYPE_CLASS.TYPE_WORD : 
		memcpy(ADR(_WORD),Source.pValue,DINT_TO_UDINT(Source.diSize));
		convertSuccessful := TryConvert_Source_TO_Destination(_WORD,_UDINT);
		
	__SYSTEM.TYPE_CLASS.TYPE_DWORD : 
		memcpy(ADR(_DWORD),Source.pValue,DINT_TO_UDINT(Source.diSize));
		convertSuccessful := TryConvert_Source_TO_Destination(_DWORD,_UDINT);
		
	__SYSTEM.TYPE_CLASS.TYPE_USINT : 
		memcpy(ADR(_USINT),Source.pValue,DINT_TO_UDINT(Source.diSize));
		convertSuccessful := TryConvert_Source_TO_Destination(_USINT,_UDINT);
		
	__SYSTEM.TYPE_CLASS.TYPE_UINT : 
		memcpy(ADR(_UINT),Source.pValue,DINT_TO_UDINT(Source.diSize));
		convertSuccessful := TryConvert_Source_TO_Destination(_UINT,_UDINT);
		
	__SYSTEM.TYPE_CLASS.TYPE_UDINT : 
		memcpy(ADR(_UDINT),Source.pValue,DINT_TO_UDINT(Source.diSize));
		convertSuccessful := TRUE;
		
ELSE 
		
	RETURN;
		
END_CASE

IF NOT convertSuccessful THEN
	RETURN;
END_IF

SetUint(jsonValue,_UDINT); // Not a typo, SetUnit actually takes a UDINT
TrySetUint := TRUE;
END_METHOD

METHOD PRIVATE TrySetUint64 : BOOL
VAR_INPUT
	JsonValue : SJsonValue;
	Source : ANY;
END_VAR
VAR
	convertSuccessful : BOOL;
	_LWORD : LWORD;
	_ULINT : ULINT;
END_VAR
CASE Source.TypeClass OF 

	__SYSTEM.TYPE_CLASS.TYPE_LWORD : 
		memcpy(ADR(_LWORD),Source.pValue,DINT_TO_UDINT(Source.diSize));
		convertSuccessful := TryConvert_Source_TO_Destination(_LWORD,_ULINT);
	
	__SYSTEM.TYPE_CLASS.TYPE_ULINT : 
		memcpy(ADR(_ULINT),Source.pValue,DINT_TO_UDINT(Source.diSize));
		convertSuccessful := TRUE;
		
ELSE 
		
	RETURN;
		
END_CASE

IF NOT convertSuccessful THEN
	RETURN;
END_IF

SetUint64(jsonValue,_ULINT);
TrySetUint64 := TRUE;
END_METHOD

METHOD PUBLIC TryLocate : BOOL
VAR_INPUT
	Path : T_MaxString;
	Destination : REFERENCE TO SJsonValue;
END_VAR
VAR
	jsonDomNavigator : JsonDomNavigator(THIS^);
	jsonPathSyntaxParser : JsonPathSyntaxParser;
	jsonValue : SJsonValue;
END_VAR
jsonPathSyntaxParser.Parse(Path, jsonDomNavigator);
jsonValue := jsonDomNavigator.CurrentNode;

IF jsonValue = 0 THEN
	RETURN;
END_IF

Destination := jsonValue;
TryLocate := TRUE;
END_METHOD

METHOD PUBLIC TryModify : BOOL
VAR_INPUT
	Path : T_MaxString;
	Source : ANY;
END_VAR
VAR
	jsonDomNavigator : JsonDomNavigator(THIS^);
	jsonPathSyntaxParser : JsonPathSyntaxParser;
	jsonValue : SJsonValue;
END_VAR
jsonPathSyntaxParser.Parse(Path, jsonDomNavigator);
jsonValue := jsonDomNavigator.CurrentNode;

IF jsonValue = 0 THEN
	RETURN;
END_IF

IF IsObject(jsonValue) THEN
	RETURN;
END_IF

IF TrySetBool(jsonValue, Source) THEN
	TryModify := TRUE;
	RETURN;
END_IF

IF TrySetString(jsonValue, Source) THEN
	TryModify := TRUE;
	RETURN;
END_IF

IF TrySetInt(jsonValue, Source) THEN
	TryModify := TRUE;
	RETURN;
END_IF

IF TrySetUint(jsonValue, Source) THEN
	TryModify := TRUE;
	RETURN;
END_IF

IF TrySetDouble(jsonValue, Source) THEN
	TryModify := TRUE;
	RETURN;
END_IF

IF TrySetInt64(jsonValue, Source) THEN
	TryModify := TRUE;
	RETURN;
END_IF

IF TrySetUint64(jsonValue, Source) THEN
	TryModify := TRUE;
	RETURN;
END_IF
END_METHOD

METHOD PUBLIC TryRead : BOOL
VAR_INPUT
	Path : T_MaxString;
	Destination : ANY;
END_VAR
VAR
	jsonDomNavigator : JsonDomNavigator(THIS^);
	jsonPathSyntaxParser : JsonPathSyntaxParser;
	jsonValue : SJsonValue;
	_BOOL : BOOL;
	_DINT : DINT;
	_LINT : LINT;
	_UDINT : UDINT;
	_ULINT : ULINT;
	_LREAL : LREAL;
	_STRING : POINTER TO STRING(1);
END_VAR
jsonPathSyntaxParser.Parse(Path, jsonDomNavigator);
jsonValue := jsonDomNavigator.CurrentNode;

IF jsonValue = 0 THEN
	RETURN;
END_IF

IF IsBool(jsonValue) THEN
	_BOOL := GetBool(jsonValue);
	TryRead := TryConvert_BOOL_TO_DESTINATION(_BOOL,Destination);
	RETURN;
END_IF

IF IsInt(jsonValue) THEN
	_DINT := GetInt(jsonValue);
	TryRead := TryConvert_DINT_TO_DESTINATION(_DINT,Destination);
	RETURN;
END_IF

IF IsInt64(jsonValue) THEN
	_LINT := GetInt64(jsonValue);
	TryRead := TryConvert_LINT_TO_DESTINATION(_LINT,Destination);
	RETURN;
END_IF

IF IsUInt(jsonValue) THEN
	_UDINT := GetUInt(jsonValue);
	TryRead := TryConvert_UDINT_TO_DESTINATION(_UDINT,Destination);
	RETURN;
END_IF

IF IsUInt64(jsonValue) THEN
	_ULINT := GetUInt64(jsonValue);
	TryRead := TryConvert_ULINT_TO_DESTINATION(_ULINT,Destination);
	RETURN;
END_IF

IF IsDouble(jsonValue) THEN
	_LREAL := GetDouble(jsonValue);
	TryRead := TryConvert_LREAL_TO_DESTINATION(_LREAL,Destination);
	RETURN;
END_IF

IF IsString(jsonValue) AND Destination.TypeClass = __SYSTEM.TYPE_CLASS.TYPE_STRING THEN
	_STRING := Destination.pValue;
	IF (CopyString(jsonValue,_STRING^,DINT_TO_UDINT(Destination.diSize)) > 0) THEN;
		TryRead := TRUE;
		RETURN;
	END_IF
END_IF
END_METHOD

METHOD PUBLIC TryWrite : BOOL
VAR_INPUT
	Path : T_MaxString;
	Source : ANY;
END_VAR
VAR
	jsonDomCreator : JsonDomCreator(THIS^);
	jsonPathSyntaxParser : JsonPathSyntaxParser;
	jsonValue : SJsonValue;
END_VAR
jsonPathSyntaxParser.Parse(Path, jsonDomCreator);
jsonValue := jsonDomCreator.CurrentNode;

IF jsonValue = 0 THEN
	RETURN;
END_IF

IF IsObject(jsonValue) THEN
	RETURN;
END_IF

IF TrySetBool(jsonValue, Source) THEN
	TryWrite := TRUE;
	RETURN;
END_IF

IF TrySetString(jsonValue, Source) THEN
	TryWrite := TRUE;
	RETURN;
END_IF

IF TrySetInt(jsonValue, Source) THEN
	TryWrite := TRUE;
	RETURN;
END_IF

IF TrySetUint(jsonValue, Source) THEN
	TryWrite := TRUE;
	RETURN;
END_IF

IF TrySetDouble(jsonValue, Source) THEN
	TryWrite := TRUE;
	RETURN;
END_IF

IF TrySetInt64(jsonValue, Source) THEN
	TryWrite := TRUE;
	RETURN;
END_IF

IF TrySetUint64(jsonValue, Source) THEN
	TryWrite := TRUE;
	RETURN;
END_IF
END_METHOD

END_FUNCTION_BLOCK

// mobject-json/_Internal/JsonPathSyntaxParser/JsonPathSyntaxParser
{attribute 'linkalways'} 
{attribute 'no_explicit_call' := 'This FB is a CLASS and must be accessed using methods or properties'}
{attribute 'enable_dynamic_creation'}
FUNCTION_BLOCK JsonPathSyntaxParser
VAR
	currentlyParsingType : (NOTHING, DOT_NOTATION_PROPERTY, BRACKET_NOTATION_PROPERTY_OR_ARRAY, BRACKET_NOTATION_PROPERTY_ELEMENT, BRACKET_NOTATION_ARRAY_ELEMENT);
END_VAR

METHOD PUBLIC Parse
VAR_INPUT
	Path : REFERENCE TO STRING;
	JsonPathVisitor : I_JsonPathVisitor;
END_VAR
VAR
	currentCharacterPositionInPath : UDINT;
	currentElementStart : UDINT;
	currentElementEnd : UDINT;
	currentElementLength : UDINT;
	elementText : T_MAXSTRING;
	endOfRepeat : BOOL;
END_VAR
VAR CONSTANT
	PERIOD : BYTE := 16#2E; // .
	DOLLAR_SIGN : BYTE := 16#24; // $
	SINGLE_QUOTE : BYTE := 16#27; // '
	LEFT_SQUARE_BRACKET : BYTE := 16#5B; // [
	RIGHT_SQUARE_BRACKET : BYTE := 16#5D; // ]
	NULL : BYTE := 0; // null
END_VAR
JsonPathVisitor.StartOfParse();

IF Path[0] = NULL THEN
	JsonPathVisitor.EndOfParse();
	RETURN;
END_IF

currentCharacterPositionInPath := 0;
currentlyParsingType := NOTHING;

REPEAT 
	
	IF Path[currentCharacterPositionInPath] = NULL THEN
		 endOfRepeat := TRUE;
	END_IF
		
	CASE currentlyParsingType OF
		
		NOTHING: 
		
			// at this point we are not currently "parsing" a known type from the string, therfore the next character should 
			// decide what type is next. 
		
			IF Path[currentCharacterPositionInPath] = DOLLAR_SIGN THEN
				
				// i.e. the following string $.myValue would indicate that we are here.
				//                           ^                                         
				// as such, we do not need to take any action.  We already create a root element at the start, so this is an 
				// optional character which they do not need to supply. 				
				
			ELSIF Path[currentCharacterPositionInPath] = PERIOD THEN
				
				// i.e. the following string $.myValue would indicate that we are here.
				//                            ^                                        
				// as such, we do not need to take any action.  
				
			ELSIF Path[currentCharacterPositionInPath] = LEFT_SQUARE_BRACKET THEN
				
				// i.e. the following string $.myValue[1].['myProperty'] would indicate that we could be at the start of one of two types
				//                                    ^   ^                                      
				// as such, we mark that we could be either a property or array and continue				
				currentlyParsingType := BRACKET_NOTATION_PROPERTY_OR_ARRAY;				
				
			ELSIF Path[currentCharacterPositionInPath] = RIGHT_SQUARE_BRACKET THEN
				
				// This would indicate a failed parse as this should not happen.
				JsonPathVisitor.InvalidSyntaxFound(RIGHT_SQUARE_BRACKET, currentCharacterPositionInPath);
				
			ELSIF Path[currentCharacterPositionInPath] = SINGLE_QUOTE THEN
				
				// This would indicate a failed parse as this should not happen.
				JsonPathVisitor.InvalidSyntaxFound(SINGLE_QUOTE, currentCharacterPositionInPath);
				
			ELSE
				
				// i.e. the following string $.myValue[1].['myProperty'] would indicate that we could be at the start of a property
				//                             ^                      
				currentlyParsingType := DOT_NOTATION_PROPERTY;
				currentElementStart := currentCharacterPositionInPath;	
		
			END_IF
			
		DOT_NOTATION_PROPERTY:
		
			IF Path[currentCharacterPositionInPath] = PERIOD OR Path[currentCharacterPositionInPath] = LEFT_SQUARE_BRACKET OR Path[currentCharacterPositionInPath] = NULL THEN
				
				currentElementEnd := currentCharacterPositionInPath - 1;
				
				currentElementLength := 1 + currentElementEnd - currentElementStart;
				memset(ADR(elementText),0,SIZEOF(elementText));
				memcpy(ADR(elementText),ADR(Path[currentElementStart]),currentElementLength);
		
				JsonPathVisitor.PropertyFound(elementText);
				
				currentlyParsingType := NOTHING;
				CONTINUE;
				
			END_IF
			
		BRACKET_NOTATION_PROPERTY_OR_ARRAY:
		
			IF Path[currentCharacterPositionInPath] = SINGLE_QUOTE THEN
				currentlyParsingType := BRACKET_NOTATION_PROPERTY_ELEMENT;
				currentElementStart := currentCharacterPositionInPath + 1;			
			ELSE
				currentlyParsingType := BRACKET_NOTATION_ARRAY_ELEMENT;
				currentElementStart := currentCharacterPositionInPath;			
			END_IF
			
		BRACKET_NOTATION_PROPERTY_ELEMENT:
		
			IF Path[currentCharacterPositionInPath] = SINGLE_QUOTE THEN
				
				currentElementEnd := currentCharacterPositionInPath - 1;

				currentElementLength := 1 + currentElementEnd - currentElementStart;
				memset(ADR(elementText),0,SIZEOF(elementText));
				memcpy(ADR(elementText),ADR(Path[currentElementStart]),currentElementLength);
				
				JsonPathVisitor.PropertyFound(elementText);
			
				currentlyParsingType := NOTHING;
						
			END_IF
			
		BRACKET_NOTATION_ARRAY_ELEMENT:
		
			IF Path[currentCharacterPositionInPath] = RIGHT_SQUARE_BRACKET THEN
				
				currentElementEnd := currentCharacterPositionInPath - 1;
				
				currentElementLength := 1 + currentElementEnd - currentElementStart;
				memset(ADR(elementText),0,SIZEOF(elementText));
				memcpy(ADR(elementText),ADR(Path[currentElementStart]),currentElementLength);
				
				JsonPathVisitor.ArrayIndexFound(STRING_TO_UDINT(elementText));		
				currentlyParsingType := NOTHING;
						
			END_IF
			

	END_CASE
	
	currentCharacterPositionInPath := currentCharacterPositionInPath + 1;
	
UNTIL endOfRepeat 
END_REPEAT

JsonPathVisitor.EndOfParse();
END_METHOD

END_FUNCTION_BLOCK

// mobject-json/_Internal/JsonPathVisitor/I_JsonPathVisitor
INTERFACE I_JsonPathVisitor EXTENDS __System.IQueryInterface

METHOD ArrayIndexFound
VAR_INPUT
	Index : UDINT;
END_VAR
END_METHOD

METHOD EndOfParse
VAR_INPUT
END_VAR
END_METHOD

METHOD InvalidSyntaxFound
VAR_INPUT
	Character : BYTE;
	Position : UDINT;
END_VAR
END_METHOD

METHOD PropertyFound
VAR_INPUT
	Name : T_MAXSTRING;
END_VAR
END_METHOD

METHOD StartOfParse
VAR_INPUT
END_VAR
END_METHOD

END_INTERFACE

// mobject-json/_Internal/JsonPathVisitor/JsonDomNavigator
{attribute 'linkalways'} 
{attribute 'no_explicit_call' := 'This FB is a CLASS and must be accessed using methods or properties'}
{attribute 'enable_dynamic_creation'}
FUNCTION_BLOCK JsonDomNavigator IMPLEMENTS I_JsonPathVisitor
VAR
	jsonDomParser : REFERENCE TO JsonDomParser;
	currentJsonPosition : SJsonValue;
	_currentNode : SJsonValue;
END_VAR

METHOD FB_init : BOOL
VAR_INPUT
	bInitRetains : BOOL; // if TRUE, the retain variables are initialized (warm start / cold start)
	bInCopyCode : BOOL;  // if TRUE, the instance afterwards gets moved into the copy code (online change)
	JsonDomParser : REFERENCE TO JsonDomParser;
END_VAR
THIS^.jsonDomParser REF= JsonDomParser;
END_METHOD

METHOD ArrayIndexFound
VAR_INPUT
	Index : UDINT;
END_VAR
currentJsonPosition := jsonDomParser.GetArrayValueByIdx(currentJsonPosition, Index);
END_METHOD

PROPERTY PUBLIC CurrentNode : SJsonValue
GET
CurrentNode := _currentNode;
END_GET
END_PROPERTY

METHOD EndOfParse
VAR_INPUT
END_VAR
_currentNode := currentJsonPosition;
END_METHOD

METHOD InvalidSyntaxFound
VAR_INPUT
	Character : BYTE;
	Position : UDINT;
END_VAR
currentJsonPosition := 0;
END_METHOD

METHOD PropertyFound
VAR_INPUT
	Name : T_MAXSTRING;
END_VAR
currentJsonPosition := jsonDomParser.FindMember(currentJsonPosition,Name);
END_METHOD

METHOD StartOfParse
VAR_INPUT
END_VAR
currentJsonPosition := jsonDomParser.GetDocumentRoot();
END_METHOD

END_FUNCTION_BLOCK

// mobject-json/_Internal/JsonPathVisitor/JsonDomCreator
{attribute 'linkalways'} 
{attribute 'no_explicit_call' := 'This FB is a CLASS and must be accessed using methods or properties'}
{attribute 'enable_dynamic_creation'}
FUNCTION_BLOCK JsonDomCreator IMPLEMENTS I_JsonPathVisitor
VAR
	jsonDomParser : REFERENCE TO JsonDomParser;
	currentJsonPosition : SJsonValue;
	_currentNode : SJsonValue;
END_VAR

METHOD FB_init : BOOL
VAR_INPUT
	bInitRetains : BOOL; // if TRUE, the retain variables are initialized (warm start / cold start)
	bInCopyCode : BOOL;  // if TRUE, the instance afterwards gets moved into the copy code (online change)
	JsonDomParser : REFERENCE TO JsonDomParser;
END_VAR
THIS^.jsonDomParser REF= JsonDomParser;
END_METHOD

METHOD PRIVATE PadStartOfArray : SJsonValue
VAR_INPUT
	Index : UDINT;
	ArrayPosition : SJsonValue;
END_VAR
VAR
	i : UDINT;
	arrayValueLocation : SJsonValue;
END_VAR
FOR i := 0 TO Index DO
		
	arrayValueLocation := jsonDomParser.GetArrayValueByIdx(ArrayPosition, Index);
	IF arrayValueLocation <> 0 THEN
		CONTINUE;
	END_IF
	
	arrayValueLocation := jsonDomParser.PushbackNullValue(ArrayPosition);

END_FOR

PadStartOfArray := arrayValueLocation;
END_METHOD

METHOD ArrayIndexFound
VAR_INPUT
	Index : UDINT;
END_VAR
VAR
	memberLocation : SJsonValue;
	i : UDINT;
END_VAR
IF jsonDomParser.IsArray(currentJsonPosition) THEN
	
	memberLocation := jsonDomParser.GetArrayValueByIdx(currentJsonPosition, Index);
	
	IF memberLocation <> 0 THEN
		currentJsonPosition := memberLocation;
		RETURN;
	END_IF
	
	currentJsonPosition := PadStartOfArray(Index, currentJsonPosition);

else
	
	memberLocation := jsonDomParser.SetArray(currentJsonPosition,0);
	currentJsonPosition := PadStartOfArray(Index, memberLocation);
	
END_IF
END_METHOD

PROPERTY PUBLIC CurrentNode : SJsonValue
GET
CurrentNode := _currentNode;
END_GET
END_PROPERTY

METHOD EndOfParse
VAR_INPUT
END_VAR
_currentNode := currentJsonPosition;
END_METHOD

METHOD InvalidSyntaxFound
VAR_INPUT
	Character : BYTE;
	Position : UDINT;
END_VAR
currentJsonPosition := 0;
END_METHOD

METHOD PropertyFound
VAR_INPUT
	Name : T_MAXSTRING;
END_VAR
VAR
	memberLocation : SJsonValue;
END_VAR
memberLocation := jsonDomParser.FindMember(currentJsonPosition,Name);

IF memberLocation <> 0 THEN
	currentJsonPosition := memberLocation;
	RETURN;
END_IF

currentJsonPosition := jsonDomParser.AddNullMember(currentJsonPosition,Name);
END_METHOD

METHOD StartOfParse
VAR_INPUT
END_VAR
currentJsonPosition := jsonDomParser.GetDocumentRoot();
END_METHOD

END_FUNCTION_BLOCK

// mobject-json/_Internal/JsonDeserializerNode/JsonDeserializerNode
{attribute 'linkalways'} 
{attribute 'no_explicit_call' := 'This FB is a CLASS and must be accessed using methods or properties'}
{attribute 'enable_dynamic_creation'}
FUNCTION_BLOCK JsonDeserializerNode EXTENDS Disposable IMPLEMENTS I_Deserializer
VAR	
	parent : I_JsonDeserializer;
	jsonParser : REFERENCE TO JsonDomParser;
	root : SJsonValue;
	garbageCollector : I_DeserializerGarbageCollector;
	nullNode : I_Deserializer;
	errorFactory : DeserializationErrorFactory;
END_VAR

METHOD FB_init : BOOL
VAR_INPUT
	bInitRetains : BOOL; // if TRUE, the retain variables are initialized (warm start / cold start)
	bInCopyCode : BOOL;  // if TRUE, the instance afterwards gets moved into the copy code (online change)
	ParentJsonDeserializer : I_JsonDeserializer;
	ParentJsonDomParser : REFERENCE TO JsonDomParser;
	NodeRoot : SJsonValue;
	ParentGarbageCollector : I_DeserializerGarbageCollector;
	ParentNullDeserializer : I_Deserializer;
END_VAR
THIS^.parent := ParentJsonDeserializer;
THIS^.jsonParser REF= ParentJsonDomParser;
THIS^.root := NodeRoot;
THIS^.garbageCollector := ParentGarbageCollector;
THIS^.nullNode := ParentNullDeserializer;

ParentGarbageCollector.Register(THIS^);
END_METHOD

METHOD PROTECTED CreateArrayForwardEnumerator : I_DeserializerArrayForwardEnumerator
VAR_INPUT
	DeserializerRoot : SJsonValue;
END_VAR
VAR 
	pForwardEnumerator : POINTER TO JsonDeserializerArrayForwardEnumerator;
END_VAR
pForwardEnumerator := __NEW(JsonDeserializerArrayForwardEnumerator(
	ParentJsonDeserializer := parent,
	ParentJsonDomParser := jsonParser, 
	NodeRoot := DeserializerRoot, 
	ParentGarbageCollector := garbageCollector, 
	ParentNullDeserializer := nullNode
));

CreateArrayForwardEnumerator := pForwardEnumerator^;
END_METHOD

METHOD PROTECTED CreateDeserializer : I_Deserializer
VAR_INPUT
	DeserializerRoot : SJsonValue;
END_VAR
VAR 
	pNode : POINTER TO JsonDeserializerNode;
END_VAR
pNode := __NEW(JsonDeserializerNode(
	ParentJsonDeserializer := parent,
	ParentJsonDomParser := jsonParser, 
	NodeRoot := DeserializerRoot, 
	ParentGarbageCollector := garbageCollector, 
	ParentNullDeserializer := nullNode
));

CreateDeserializer := pNode^;
END_METHOD

METHOD PROTECTED CreateObjectForwardEnumerator : I_DeserializerObjectForwardEnumerator
VAR_INPUT
	DeserializerRoot : SJsonValue;
END_VAR
VAR 
	pForwardEnumerator : POINTER TO JsonDeserializerObjectForwardEnumerator;
END_VAR
pForwardEnumerator := __NEW(JsonDeserializerObjectForwardEnumerator(
	ParentJsonDeserializer := parent,
	ParentJsonDomParser := jsonParser, 
	NodeRoot := DeserializerRoot, 
	ParentGarbageCollector := garbageCollector, 
	ParentNullDeserializer := nullNode
));

CreateObjectForwardEnumerator := pForwardEnumerator^;
END_METHOD

METHOD PROTECTED TryGetMember : BOOL
VAR_INPUT
	MemberName : T_MAXSTRING;
	Member : REFERENCE TO SJsonValue;
	Feedback : I_DeserializerFeedback;
END_VAR
VAR
	localMember : SJsonValue;
	error : I_Error;
END_VAR
IF MemberName = '' THEN
	error := errorFactory.CreateInvalidKeyError();
	Feedback.LogError(error);
	RETURN;
END_IF

localMember := jsonParser.FindMember(root, MemberName);

IF localMember = 0 THEN
	error := errorFactory.CreateMissingKeyError(MemberName);
	Feedback.LogError(error);
	RETURN;
END_IF

Member := localMember;
TryGetMember := TRUE;
END_METHOD

METHOD PROTECTED TryReadBool : BOOL
VAR_INPUT
	JsonValue : SJsonValue;
	Destination : ANY;
END_VAR
VAR
	_BOOL : BOOL;
END_VAR
IF jsonValue = 0 THEN
	RETURN;
END_IF

IF jsonParser.IsBool(jsonValue) THEN
	_BOOL := jsonParser.GetBool(jsonValue);
	TryReadBool := TryConvert_BOOL_TO_DESTINATION(_BOOL,Destination);
	RETURN;
END_IF
END_METHOD

METHOD PROTECTED TryReadNumber : BOOL
VAR_INPUT
	JsonValue : SJsonValue;
	Destination : ANY;
END_VAR
VAR
	_DINT : DINT;
	_LINT : LINT;
	_UDINT : UDINT;
	_ULINT : ULINT;
	_LREAL : LREAL;
END_VAR
IF jsonValue = 0 THEN
	RETURN;
END_IF

IF jsonParser.IsInt(jsonValue) THEN
	_DINT := jsonParser.GetInt(jsonValue);
	TryReadNumber := TryConvert_DINT_TO_DESTINATION(_DINT,Destination);
	RETURN;
END_IF

IF jsonParser.IsInt64(jsonValue) THEN
	_LINT := jsonParser.GetInt64(jsonValue);
	TryReadNumber := TryConvert_LINT_TO_DESTINATION(_LINT,Destination);
	RETURN;
END_IF

IF jsonParser.IsUInt(jsonValue) THEN
	_UDINT := jsonParser.GetUInt(jsonValue);
	TryReadNumber := TryConvert_UDINT_TO_DESTINATION(_UDINT,Destination);
	RETURN;
END_IF

IF jsonParser.IsUInt64(jsonValue) THEN
	_ULINT := jsonParser.GetUInt64(jsonValue);
	TryReadNumber := TryConvert_ULINT_TO_DESTINATION(_ULINT,Destination);
	RETURN;
END_IF

IF jsonParser.IsDouble(jsonValue) THEN
	_LREAL := jsonParser.GetDouble(jsonValue);
	TryReadNumber := TryConvert_LREAL_TO_DESTINATION(_LREAL,Destination);
	RETURN;
END_IF
END_METHOD

METHOD PROTECTED TryReadString : BOOL
VAR_INPUT
	JsonValue : SJsonValue;
	Destination : REFERENCE TO T_MAXSTRING;
END_VAR
IF jsonValue = 0 THEN
	RETURN;
END_IF

IF jsonParser.IsString(jsonValue) THEN
	IF (jsonParser.CopyString(jsonValue,Destination,DINT_TO_UDINT(SIZEOF(Destination))) > 0) THEN;
		TryReadString := TRUE;
		RETURN;
	END_IF
END_IF
END_METHOD

METHOD PROTECTED TryReadStringEx : BOOL
VAR_INPUT
	JsonValue : SJsonValue;
	DestinationAddress : POINTER TO STRING;
	DestinationSize : UDINT;
END_VAR
IF jsonValue = 0 THEN
	RETURN;
END_IF

IF jsonParser.IsString(jsonValue) THEN
	IF (jsonParser.CopyString(jsonValue,DestinationAddress^,DestinationSize) > 0) THEN;
		TryReadStringEx := TRUE;
		RETURN;
	END_IF
END_IF
END_METHOD

METHOD PUBLIC Clone : I_Deserializer
VAR
	pClone : POINTER TO JsonDeserializer;
	jsonSize : UDINT;
	pJsonString : POINTER TO STRING;
END_VAR
pClone := __NEW(JsonDeserializer);
Clone := pClone^;

jsonSize := jsonParser.GetJsonLength(root);

IF jsonSize = 0 THEN
	// no further cloning to do. 
	RETURN;
END_IF

pJsonString := __NEW(BYTE, jsonSize);

IF jsonParser.CopyJson(root, pJsonString^, jsonSize) = 0 THEN
	__DELETE(pJsonString);
	RETURN;
END_IF

pClone^.TryLoad(pJsonString^);
__DELETE(pJsonString);
END_METHOD

METHOD Dispose
VAR
END_VAR
garbageCollector.Deregister(THIS^);
super^.Dispose();
END_METHOD

METHOD GetArray : I_Deserializer
IF NOT jsonParser.IsArray(root) THEN
	GetArray := nullNode;
	RETURN;
END_IF

GetArray := CreateDeserializer(root);
END_METHOD

METHOD GetArrayEnumerator : I_DeserializerArrayForwardEnumerator
VAR_INPUT
END_VAR
GetArrayEnumerator := CreateArrayForwardEnumerator(root);
END_METHOD

METHOD GetElementByIndex : I_Deserializer
VAR_INPUT
	Index : UDINT;
END_VAR
VAR
	newRoot : SJsonValue;
END_VAR
IF NOT jsonParser.IsArray(root) THEN
	GetElementByIndex := nullNode;
	RETURN;
END_IF

newRoot := jsonParser.GetArrayValueByIdx(root, Index);

IF newRoot = 0 THEN
	GetElementByIndex := nullNode;
	RETURN;
END_IF

GetElementByIndex := CreateDeserializer(newRoot);
END_METHOD

METHOD GetKeyArray : I_Deserializer
VAR_INPUT
	Key : T_MAXSTRING;
END_VAR
VAR
	member : SJsonValue;
END_VAR
IF key = '' THEN
	RETURN;
END_IF

member := jsonParser.FindMember(root,Key);

IF member = 0 THEN
	GetKeyArray := nullNode;
	RETURN;
END_IF

IF NOT jsonParser.IsArray(member) THEN
	GetKeyArray := nullNode;
	RETURN;
END_IF

GetKeyArray := CreateDeserializer(member);
END_METHOD

METHOD GetKeyObject : I_Deserializer
VAR_INPUT
	Key : T_MAXSTRING;
END_VAR
VAR
	newRoot : SJsonValue;
END_VAR
newRoot := jsonParser.FindMember(root, Key);

IF newRoot = 0 THEN
	GetKeyObject := nullNode;
	RETURN;
END_IF

GetKeyObject := CreateDeserializer(newRoot);
END_METHOD

METHOD GetObject : I_Deserializer
IF NOT jsonParser.IsObject(root) THEN
	GetObject := nullNode;
	RETURN;
END_IF

GetObject := CreateDeserializer(root);
END_METHOD

METHOD GetObjectEnumerator : I_DeserializerObjectForwardEnumerator
VAR_INPUT
END_VAR
GetObjectEnumerator := CreateObjectForwardEnumerator(root);
END_METHOD

METHOD GetValue : I_Deserializer
VAR
	newRoot : SJsonValue;
END_VAR
newRoot := jsonParser.GetMemberValue(root);

IF newRoot = 0 THEN
	GetValue := nullNode;
	RETURN;
END_IF

GetValue := CreateDeserializer(newRoot);
END_METHOD

METHOD TryDeserializeKeyToObject : BOOL
VAR_INPUT
	Key : T_MAXSTRING;
	Object : I_Deserializable;
	Feedback : I_DeserializerFeedback;
END_VAR
VAR
	member : SJsonValue;
	error : I_Error;
	deserializer : I_Deserializer;
END_VAR
IF NOT TryGetMember(Key, member, Feedback) THEN
	RETURN;
END_IF

deserializer := CreateDeserializer(member);
TryDeserializeKeyToObject := Object.TryDeserializeFrom(deserializer, Feedback);
END_METHOD

METHOD TryDeserializeToObject : BOOL
VAR_INPUT
	Object : I_Deserializable;
	Feedback : I_DeserializerFeedback;
END_VAR
TryDeserializeToObject := Object.TryDeserializeFrom(THIS^, Feedback);
END_METHOD

METHOD TryGetBase64 : BOOL
VAR_INPUT
	pBytes : POINTER TO BYTE;
	nBytes : DINT;
	Feedback : I_DeserializerFeedback;
END_VAR
VAR
	error : I_Error;
END_VAR
IF NOT jsonParser.IsBase64(root) THEN
	error := errorFactory.CreateIncorrectTypeError('Base64');
	Feedback.LogError(error);
	RETURN;
END_IF

jsonParser.GetBase64(root, pBytes, nBytes);
TryGetBase64 := TRUE;
END_METHOD

METHOD TryGetBool : BOOL
VAR_INPUT
	Destination : REFERENCE TO BOOL;
	Feedback : I_DeserializerFeedback;
END_VAR
VAR
	value : BOOL;
	error : I_Error;
END_VAR
IF NOT TryReadBool(root, value) THEN
	error := errorFactory.CreateIncorrectTypeError('BOOL');
	Feedback.LogError(error);
	RETURN;
END_IF

Destination := value;
TryGetBool := TRUE;
END_METHOD

METHOD TryGetByte : BOOL
VAR_INPUT
	Destination : REFERENCE TO BYTE;
	Feedback : I_DeserializerFeedback;
END_VAR
VAR
	value : BYTE;
	error : I_Error;
END_VAR
IF NOT TryReadNumber(root, value) THEN
	error := errorFactory.CreateIncorrectTypeError('BYTE');
	Feedback.LogError(error);
	RETURN;
END_IF

Destination := value;
TryGetByte := TRUE;
END_METHOD

METHOD TryGetDateTime : BOOL
VAR_INPUT
	Destination : REFERENCE TO DATE_AND_TIME;
	Feedback : I_DeserializerFeedback;
END_VAR
VAR
	error : I_Error;
END_VAR
IF NOT jsonParser.IsISO8601TimeFormat(root) THEN
	error := errorFactory.CreateIncorrectTypeError('DATE_AND_TIME');
	Feedback.LogError(error);
	RETURN;
END_IF

Destination := jsonParser.GetDateTime(root);
TryGetDateTime := TRUE;
END_METHOD

METHOD TryGetDcTime : BOOL
VAR_INPUT
	Destination : REFERENCE TO DCTIME;
	Feedback : I_DeserializerFeedback;
END_VAR
VAR
	error : I_Error;
END_VAR
IF NOT jsonParser.IsISO8601TimeFormat(root) THEN
	error := errorFactory.CreateIncorrectTypeError('DCTIME');
	Feedback.LogError(error);
	RETURN;
END_IF

Destination := jsonParser.GetDcTime(root);
TryGetDcTime := TRUE;
END_METHOD

METHOD TryGetDint : BOOL
VAR_INPUT
	Destination : REFERENCE TO DINT;
	Feedback : I_DeserializerFeedback;
END_VAR
VAR
	value : DINT;
	error : I_Error;
END_VAR
IF NOT TryReadNumber(root, value) THEN
	error := errorFactory.CreateIncorrectTypeError('DINT');
	Feedback.LogError(error);
	RETURN;
END_IF

Destination := value;
TryGetDint := TRUE;
END_METHOD

METHOD TryGetDword : BOOL
VAR_INPUT
	Destination : REFERENCE TO DWORD;
	Feedback : I_DeserializerFeedback;
END_VAR
VAR
	value : DWORD;
	error : I_Error;
END_VAR
IF NOT TryReadNumber(root, value) THEN
	error := errorFactory.CreateIncorrectTypeError('DWORD');
	Feedback.LogError(error);
	RETURN;
END_IF

Destination := value;
TryGetDword := TRUE;
END_METHOD

METHOD TryGetElementByIndex : BOOL
VAR_INPUT
	Index : UDINT;
	Destination : REFERENCE TO I_Deserializer;
	Feedback : I_DeserializerFeedback;
END_VAR
VAR
	newRoot : SJsonValue;
	error : I_Error;
END_VAR
IF NOT jsonParser.IsArray(root) THEN
	error := errorFactory.CreateIncorrectTypeError('ARRAY');
	Feedback.LogError(error);
	RETURN;
END_IF

newRoot := jsonParser.GetArrayValueByIdx(root, Index);

IF newRoot = 0 THEN
	error := errorFactory.CreateInvalidArrayIndexError(Index);
	Feedback.LogError(error);
	RETURN;
END_IF

Destination := CreateDeserializer(newRoot);
TryGetElementByIndex := TRUE;
END_METHOD

METHOD TryGetFileTime : BOOL
VAR_INPUT
	Destination : REFERENCE TO FILETIME;
	Feedback : I_DeserializerFeedback;
END_VAR
VAR
	error : I_Error;
END_VAR
IF NOT jsonParser.IsISO8601TimeFormat(root) THEN
	error := errorFactory.CreateIncorrectTypeError('FILETIME');
	Feedback.LogError(error);
	RETURN;
END_IF

Destination := jsonParser.GetFileTime(root);
TryGetFileTime := TRUE;
END_METHOD

METHOD TryGetHexAsBytes : BOOL
VAR_INPUT
	pBytes : POINTER TO BYTE;
	nBytes : DINT;
	Feedback : I_DeserializerFeedback;
END_VAR
VAR
	error : I_Error;
END_VAR
IF NOT jsonParser.IsHexBinary(root) THEN
	error := errorFactory.CreateIncorrectTypeError('HexBinary');
	Feedback.LogError(error);
	RETURN;
END_IF

jsonParser.GetHexBinary(root, pBytes, nBytes);
TryGetHexAsBytes := TRUE;
END_METHOD

METHOD TryGetInt : BOOL
VAR_INPUT
	Destination : REFERENCE TO INT;
	Feedback : I_DeserializerFeedback;
END_VAR
VAR
	value : INT;
	error : I_Error;
END_VAR
IF NOT TryReadNumber(root, value) THEN
	error := errorFactory.CreateIncorrectTypeError('INT');
	Feedback.LogError(error);
	RETURN;
END_IF

Destination := value;
TryGetInt := TRUE;
END_METHOD

METHOD TryGetKeyBase64 : BOOL
VAR_INPUT
	Key : T_MAXSTRING;
	pBytes : POINTER TO BYTE;
	nBytes : DINT;
	Feedback : I_DeserializerFeedback;
END_VAR
VAR
	member : SJsonValue;
	error : I_Error;
END_VAR
IF NOT TryGetMember(Key, member, Feedback) THEN
	RETURN;
END_IF

IF NOT jsonParser.IsBase64(member) THEN
	error := errorFactory.CreateIncorrectKeyTypeError('Base64',Key);
	Feedback.LogError(error);
	RETURN;
END_IF

jsonParser.GetBase64(member, pBytes, nBytes);
TryGetKeyBase64 := TRUE;
END_METHOD

METHOD TryGetKeyBool : BOOL
VAR_INPUT
	Key : T_MAXSTRING;
	Destination : REFERENCE TO BOOL;
	Feedback : I_DeserializerFeedback;
END_VAR
VAR
	member : SJsonValue;
	value : BOOL;
	error : I_Error;
END_VAR
IF NOT TryGetMember(Key, member, Feedback) THEN
	RETURN;
END_IF

IF NOT TryReadBool(member, value) THEN
	error := errorFactory.CreateIncorrectKeyTypeError('BOOL',Key);
	Feedback.LogError(error);
	RETURN;
END_IF

Destination := value;
TryGetKeyBool := TRUE;
END_METHOD

METHOD TryGetKeyByte : BOOL
VAR_INPUT
	Key : T_MAXSTRING;
	Destination : REFERENCE TO BYTE;
	Feedback : I_DeserializerFeedback;
END_VAR
VAR
	value : BYTE;
	member : SJsonValue;
	error : I_Error;
END_VAR
IF NOT TryGetMember(Key, member, Feedback) THEN
	RETURN;
END_IF

IF NOT TryReadNumber(member, value) THEN
	error := errorFactory.CreateIncorrectKeyTypeError('BYTE',Key);
	Feedback.LogError(error);
	RETURN;
END_IF

Destination := value;
TryGetKeyByte := TRUE;
END_METHOD

METHOD TryGetKeyDateTime : BOOL
VAR_INPUT
	Key : T_MAXSTRING;
	Destination : REFERENCE TO DATE_AND_TIME;
	Feedback : I_DeserializerFeedback;
END_VAR
VAR
	member : SJSonValue;
	error : I_Error;
END_VAR
IF NOT TryGetMember(Key, member, Feedback) THEN
	RETURN;
END_IF

IF NOT jsonParser.IsISO8601TimeFormat(member) THEN
	error := errorFactory.CreateIncorrectKeyTypeError('DATE_AND_TIME',Key);
	Feedback.LogError(error);
	RETURN;
END_IF

Destination := jsonParser.GetDateTime(member);
TryGetKeyDateTime := TRUE;
END_METHOD

METHOD TryGetKeyDcTime : BOOL
VAR_INPUT
	Key : T_MAXSTRING;
	Destination : REFERENCE TO DCTIME;
	Feedback : I_DeserializerFeedback;
END_VAR
VAR
	member : SJSonValue;
	error : I_Error;
END_VAR
IF NOT TryGetMember(Key, member, Feedback) THEN
	RETURN;
END_IF

IF NOT jsonParser.IsISO8601TimeFormat(member) THEN
	error := errorFactory.CreateIncorrectKeyTypeError('DCTIME',Key);
	Feedback.LogError(error);
	RETURN;
END_IF

Destination := jsonParser.GetDcTime(member);
TryGetKeyDcTime := TRUE;
END_METHOD

METHOD TryGetKeyDint : BOOL
VAR_INPUT
	Key : T_MAXSTRING;
	Destination : REFERENCE TO DINT;
	Feedback : I_DeserializerFeedback;
END_VAR
VAR
	member : SJsonValue;
	value : DINT;
	error : I_Error;
END_VAR
IF NOT TryGetMember(Key, member, Feedback) THEN
	RETURN;
END_IF

IF NOT TryReadNumber(member, value) THEN
	error := errorFactory.CreateIncorrectKeyTypeError('DINT',Key);
	Feedback.LogError(error);
	RETURN;
END_IF

Destination := value;
TryGetKeyDint := TRUE;
END_METHOD

METHOD TryGetKeyDword : BOOL
VAR_INPUT
	Key : T_MAXSTRING;
	Destination : REFERENCE TO DWORD;
	Feedback : I_DeserializerFeedback;
END_VAR
VAR
	member : SJsonValue;
	value : DWORD;
	error : I_Error;
END_VAR
IF NOT TryGetMember(Key, member, Feedback) THEN
	RETURN;
END_IF

IF NOT TryReadNumber(member, value) THEN
	error := errorFactory.CreateIncorrectKeyTypeError('DWORD',Key);
	Feedback.LogError(error);
	RETURN;
END_IF

Destination := value;
TryGetKeyDword := TRUE;
END_METHOD

METHOD TryGetKeyFileTime : BOOL
VAR_INPUT
	Key : T_MAXSTRING;
	Destination : REFERENCE TO FILETIME;
	Feedback : I_DeserializerFeedback;
END_VAR
VAR
	member : SJSonValue;
	error : I_Error;
END_VAR
IF NOT TryGetMember(Key, member, Feedback) THEN
	RETURN;
END_IF

IF NOT jsonParser.IsISO8601TimeFormat(member) THEN
	error := errorFactory.CreateIncorrectKeyTypeError('FILETIME',Key);
	Feedback.LogError(error);
	RETURN;
END_IF

Destination := jsonParser.GetFileTime(member);
TryGetKeyFileTime := TRUE;
END_METHOD

METHOD TryGetKeyHexAsBytes : BOOL
VAR_INPUT
	Key : T_MAXSTRING;
	pBytes : POINTER TO BYTE;
	nBytes : DINT;
	Feedback : I_DeserializerFeedback;
END_VAR
VAR
	member : SJsonValue;
	error : I_Error;
END_VAR
IF NOT TryGetMember(Key, member, Feedback) THEN
	RETURN;
END_IF

IF NOT jsonParser.IsHexBinary(member) THEN
	error := errorFactory.CreateIncorrectKeyTypeError('HexBinary',Key);
	Feedback.LogError(error);
	RETURN;
END_IF

jsonParser.GetHexBinary(member, pBytes, nBytes);
TryGetKeyHexAsBytes := TRUE;
END_METHOD

METHOD TryGetKeyInt : BOOL
VAR_INPUT
	Key : T_MAXSTRING;
	Destination : REFERENCE TO INT;
	Feedback : I_DeserializerFeedback;
END_VAR
VAR
	member : SJsonValue;
	value : INT;
	error : I_Error;
END_VAR
IF NOT TryGetMember(Key, member, Feedback) THEN
	RETURN;
END_IF

IF NOT TryReadNumber(member, value) THEN
	error := errorFactory.CreateIncorrectKeyTypeError('INT',Key);
	Feedback.LogError(error);
	RETURN;
END_IF

Destination := value;
TryGetKeyInt := TRUE;
END_METHOD

METHOD TryGetKeyLint : BOOL
VAR_INPUT
	Key : T_MAXSTRING;
	Destination : REFERENCE TO LINT;
	Feedback : I_DeserializerFeedback;
END_VAR
VAR
	member : SJsonValue;
	value : LINT;
	error : I_Error;
END_VAR
IF NOT TryGetMember(Key, member, Feedback) THEN
	RETURN;
END_IF

IF NOT TryReadNumber(member, value) THEN
	error := errorFactory.CreateIncorrectKeyTypeError('LINT',Key);
	Feedback.LogError(error);
	RETURN;
END_IF

Destination := value;
TryGetKeyLint := TRUE;
END_METHOD

METHOD TryGetKeyLreal : BOOL
VAR_INPUT
	Key : T_MAXSTRING;
	Destination : REFERENCE TO LREAL;
	Feedback : I_DeserializerFeedback;
END_VAR
VAR
	member : SJsonValue;
	value : LREAL;
	error : I_Error;
END_VAR
IF NOT TryGetMember(Key, member, Feedback) THEN
	RETURN;
END_IF

IF NOT TryReadNumber(member, value) THEN
	error := errorFactory.CreateIncorrectKeyTypeError('LREAL',Key);
	Feedback.LogError(error);
	RETURN;
END_IF

Destination := value;
TryGetKeyLreal := TRUE;
END_METHOD

METHOD TryGetKeyLtime : BOOL
VAR_INPUT
	Key : T_MAXSTRING;
	Destination : REFERENCE TO LTIME;
	Feedback : I_DeserializerFeedback;
END_VAR
VAR
	member : SJsonValue;
	timeAsString : T_MAXSTRING;
	error : I_Error;
END_VAR
IF NOT TryGetMember(Key, member, Feedback) THEN
	RETURN;
END_IF

IF NOT jsonParser.IsString(member) THEN
	error := errorFactory.CreateIncorrectKeyTypeError('LTIME',Key);
	Feedback.LogError(error);
	RETURN;
END_IF

timeAsString := jsonParser.GetString(member);
Destination := STRING_TO_LTIME(timeAsString);

TryGetKeyLtime := TRUE;
END_METHOD

METHOD TryGetKeyLword : BOOL
VAR_INPUT
	Key : T_MAXSTRING;
	Destination : REFERENCE TO LWORD;
	Feedback : I_DeserializerFeedback;
END_VAR
VAR
	member : SJsonValue;
	value : LWORD;
	error : I_Error;
END_VAR
IF NOT TryGetMember(Key, member, Feedback) THEN
	RETURN;
END_IF

IF NOT TryReadNumber(member, value) THEN
	error := errorFactory.CreateIncorrectKeyTypeError('LWORD',Key);
	Feedback.LogError(error);
	RETURN;
END_IF

Destination := value;
TryGetKeyLword := TRUE;
END_METHOD

METHOD TryGetKeyReal : BOOL
VAR_INPUT
	Key : T_MAXSTRING;
	Destination : REFERENCE TO REAL;
	Feedback : I_DeserializerFeedback;
END_VAR
VAR
	member : SJsonValue;
	value : REAL;
	error : I_Error;
END_VAR
IF NOT TryGetMember(Key, member, Feedback) THEN
	RETURN;
END_IF

IF NOT TryReadNumber(member, value) THEN
	error := errorFactory.CreateIncorrectKeyTypeError('REAL',Key);
	Feedback.LogError(error);
	RETURN;
END_IF

Destination := value;
TryGetKeyReal := TRUE;
END_METHOD

METHOD TryGetKeySint : BOOL
VAR_INPUT
	Key : T_MAXSTRING;
	Destination : REFERENCE TO SINT;
	Feedback : I_DeserializerFeedback;
END_VAR
VAR
	member : SJsonValue;
	value : SINT;
	error : I_Error;
END_VAR
IF NOT TryGetMember(Key, member, Feedback) THEN
	RETURN;
END_IF

IF NOT TryReadNumber(member, value) THEN
	error := errorFactory.CreateIncorrectKeyTypeError('SINT',Key);
	Feedback.LogError(error);
	RETURN;
END_IF

Destination := value;
TryGetKeySint := TRUE;
END_METHOD

METHOD TryGetKeyString : BOOL
VAR_INPUT
	Key : T_MAXSTRING;
	Destination : REFERENCE TO T_MAXSTRING;
	Feedback : I_DeserializerFeedback;
END_VAR
VAR
	member : SJsonValue;
	error : I_Error;
END_VAR
IF NOT TryGetMember(Key, member, Feedback) THEN
	RETURN;
END_IF

IF NOT TryReadString(member, Destination) THEN
	error := errorFactory.CreateIncorrectKeyTypeError('STRING',Key);
	Feedback.LogError(error);
	RETURN;
END_IF

TryGetKeyString := TRUE;
END_METHOD

METHOD TryGetKeyStringEx : BOOL
VAR_INPUT
	Key : T_MAXSTRING;
	DestinationAddress : POINTER TO STRING;
	DestinationSize : UDINT;
	Feedback : I_DeserializerFeedback;
END_VAR
VAR
	member : SJsonValue;
	error : I_Error;
END_VAR
IF NOT TryGetMember(Key, member, Feedback) THEN
	RETURN;
END_IF

IF NOT TryReadStringEx(member, DestinationAddress, DestinationSize) THEN
	error := errorFactory.CreateIncorrectKeyTypeError('STRING',Key);
	Feedback.LogError(error);
	RETURN;
END_IF

TryGetKeyStringEx := TRUE;
END_METHOD

METHOD TryGetKeyTime : BOOL
VAR_INPUT
	Key : T_MAXSTRING;
	Destination : REFERENCE TO TIME;
	Feedback : I_DeserializerFeedback;
END_VAR
VAR
	member : SJsonValue;
	timeAsString : T_MAXSTRING;
	error : I_Error;
END_VAR
IF NOT TryGetMember(Key, member, Feedback) THEN
	RETURN;
END_IF

IF NOT jsonParser.IsString(member) THEN
	error := errorFactory.CreateIncorrectKeyTypeError('TIME',Key);
	Feedback.LogError(error);
	RETURN;
END_IF

timeAsString := jsonParser.GetString(member);
Destination := STRING_TO_TIME(timeAsString);

TryGetKeyTime := TRUE;
END_METHOD

METHOD TryGetKeyTod : BOOL
VAR_INPUT
	Key : T_MAXSTRING;
	Destination : REFERENCE TO TOD;
	Feedback : I_DeserializerFeedback;
END_VAR
VAR
	member : SJsonValue;
	timeAsString : T_MAXSTRING;
	error : I_Error;
END_VAR
IF NOT TryGetMember(Key, member, Feedback) THEN
	RETURN;
END_IF

IF NOT jsonParser.IsString(member) THEN
	error := errorFactory.CreateIncorrectKeyTypeError('TOD',Key);
	Feedback.LogError(error);
	RETURN;
END_IF

timeAsString := jsonParser.GetString(member);
Destination := STRING_TO_TOD(timeAsString);

TryGetKeyTod := TRUE;
END_METHOD

METHOD TryGetKeyUdint : BOOL
VAR_INPUT
	Key : T_MAXSTRING;
	Destination : REFERENCE TO UDINT;
	Feedback : I_DeserializerFeedback;
END_VAR
VAR
	member : SJsonValue;
	value : UDINT;
	error : I_Error;
END_VAR
IF NOT TryGetMember(Key, member, Feedback) THEN
	RETURN;
END_IF

IF NOT TryReadNumber(member, value) THEN
	error := errorFactory.CreateIncorrectKeyTypeError('UDINT',Key);
	Feedback.LogError(error);
	RETURN;
END_IF

Destination := value;
TryGetKeyUdint := TRUE;
END_METHOD

METHOD TryGetKeyUint : BOOL
VAR_INPUT
	Key : T_MAXSTRING;
	Destination : REFERENCE TO UINT;
	Feedback : I_DeserializerFeedback;
END_VAR
VAR
	member : SJsonValue;
	value : UINT;
	error : I_Error;
END_VAR
IF NOT TryGetMember(Key, member, Feedback) THEN
	RETURN;
END_IF

IF NOT TryReadNumber(member, value) THEN
	error := errorFactory.CreateIncorrectKeyTypeError('UINT',Key);
	Feedback.LogError(error);
	RETURN;
END_IF

Destination := value;
TryGetKeyUint := TRUE;
END_METHOD

METHOD TryGetKeyUlint : BOOL
VAR_INPUT
	Key : T_MAXSTRING;
	Destination : REFERENCE TO ULINT;
	Feedback : I_DeserializerFeedback;
END_VAR
VAR
	member : SJsonValue;
	value : ULINT;
	error : I_Error;
END_VAR
IF NOT TryGetMember(Key, member, Feedback) THEN
	RETURN;
END_IF

IF NOT TryReadNumber(member, value) THEN
	error := errorFactory.CreateIncorrectKeyTypeError('ULINT',Key);
	Feedback.LogError(error);
	RETURN;
END_IF

Destination := value;
TryGetKeyUlint := TRUE;
END_METHOD

METHOD TryGetKeyUsint : BOOL
VAR_INPUT
	Key : T_MAXSTRING;
	Destination : REFERENCE TO USINT;
	Feedback : I_DeserializerFeedback;
END_VAR
VAR
	member : SJsonValue;
	value : USINT;
	error : I_Error;
END_VAR
IF NOT TryGetMember(Key, member, Feedback) THEN
	RETURN;
END_IF

IF NOT TryReadNumber(member, value) THEN
	error := errorFactory.CreateIncorrectKeyTypeError('USINT',Key);
	Feedback.LogError(error);
	RETURN;
END_IF

Destination := value;
TryGetKeyUsint := TRUE;
END_METHOD

METHOD TryGetKeyWord : BOOL
VAR_INPUT
	Key : T_MAXSTRING;
	Destination : REFERENCE TO WORD;
	Feedback : I_DeserializerFeedback;
END_VAR
VAR
	member : SJsonValue;
	value : WORD;
	error : I_Error;
END_VAR
IF NOT TryGetMember(Key, member, Feedback) THEN
	RETURN;
END_IF

IF NOT TryReadNumber(member, value) THEN
	error := errorFactory.CreateIncorrectKeyTypeError('USINT',Key);
	Feedback.LogError(error);
	RETURN;
END_IF

Destination := value;
TryGetKeyWord := TRUE;
END_METHOD

METHOD TryGetLint : BOOL
VAR_INPUT
	Destination : REFERENCE TO LINT;
	Feedback : I_DeserializerFeedback;
END_VAR
VAR
	value : LINT;
	error : I_Error;
END_VAR
IF NOT TryReadNumber(root, value) THEN
	error := errorFactory.CreateIncorrectTypeError('LINT');
	Feedback.LogError(error);
	RETURN;
END_IF

Destination := value;
TryGetLint := TRUE;
END_METHOD

METHOD TryGetLreal : BOOL
VAR_INPUT
	Destination : REFERENCE TO LREAL;
	Feedback : I_DeserializerFeedback;
END_VAR
VAR
	value : LREAL;
	error : I_Error;
END_VAR
IF NOT TryReadNumber(root, value) THEN
	error := errorFactory.CreateIncorrectTypeError('LREAL');
	Feedback.LogError(error);
	RETURN;
END_IF

Destination := value;
TryGetLreal := TRUE;
END_METHOD

METHOD TryGetLtime : BOOL
VAR_INPUT
	Destination : REFERENCE TO LTIME;
	Feedback : I_DeserializerFeedback;
END_VAR
VAR
	timeAsString : T_MAXSTRING;
	error : I_Error;
END_VAR
IF NOT jsonParser.IsString(root) THEN
	error := errorFactory.CreateIncorrectTypeError('LTIME');
	Feedback.LogError(error);
	RETURN;
END_IF

timeAsString := jsonParser.GetString(root);
Destination := STRING_TO_LTIME(timeAsString);

TryGetLtime := TRUE;
END_METHOD

METHOD TryGetLword : BOOL
VAR_INPUT
	Destination : REFERENCE TO LWORD;
	Feedback : I_DeserializerFeedback;
END_VAR
VAR
	value : LWORD;
	error : I_Error;
END_VAR
IF NOT TryReadNumber(root, value) THEN
	error := errorFactory.CreateIncorrectTypeError('LWORD');
	Feedback.LogError(error);
	RETURN;
END_IF

Destination := value;
TryGetLword := TRUE;
END_METHOD

METHOD TryGetReal : BOOL
VAR_INPUT
	Destination : REFERENCE TO REAL;
	Feedback : I_DeserializerFeedback;
END_VAR
VAR
	value : REAL;
	error : I_Error;
END_VAR
IF NOT TryReadNumber(root, value) THEN
	error := errorFactory.CreateIncorrectTypeError('REAL');
	Feedback.LogError(error);
	RETURN;
END_IF

Destination := value;
TryGetReal := TRUE;
END_METHOD

METHOD TryGetSint : BOOL
VAR_INPUT
	Destination : REFERENCE TO SINT;
	Feedback : I_DeserializerFeedback;
END_VAR
VAR
	value : SINT;
	error : I_Error;
END_VAR
IF NOT TryReadNumber(root, value) THEN
	error := errorFactory.CreateIncorrectTypeError('SINT');
	Feedback.LogError(error);
	RETURN;
END_IF

Destination := value;
TryGetSint := TRUE;
END_METHOD

METHOD TryGetString : BOOL
VAR_INPUT
	Destination : REFERENCE TO T_MAXSTRING;
	Feedback : I_DeserializerFeedback;
END_VAR
VAR
	error : I_Error;
END_VAR
IF NOT TryReadString(root, Destination) THEN
	error := errorFactory.CreateIncorrectTypeError('STRING');
	Feedback.LogError(error);
	RETURN;
END_IF

TryGetString := TRUE;
END_METHOD

METHOD TryGetStringEx : BOOL
VAR_INPUT
	DestinationAddress : POINTER TO STRING;
	DestinationSize : UDINT;
	Feedback : I_DeserializerFeedback;
END_VAR
VAR
	error : I_Error;
END_VAR
IF NOT TryReadStringEx(root, DestinationAddress, DestinationSize) THEN
	error := errorFactory.CreateIncorrectTypeError('STRING');
	Feedback.LogError(error);
	RETURN;
END_IF

TryGetStringEx := TRUE;
END_METHOD

METHOD TryGetTime : BOOL
VAR_INPUT
	Destination : REFERENCE TO TIME;
	Feedback : I_DeserializerFeedback;
END_VAR
VAR
	timeAsString : T_MAXSTRING;
	error : I_Error;
END_VAR
IF NOT jsonParser.IsString(root) THEN
	error := errorFactory.CreateIncorrectTypeError('TIME');
	Feedback.LogError(error);
	RETURN;
END_IF

timeAsString := jsonParser.GetString(root);
Destination := STRING_TO_TIME(timeAsString);

TryGetTime := TRUE;
END_METHOD

METHOD TryGetTod : BOOL
VAR_INPUT
	Destination : REFERENCE TO TOD;
	Feedback : I_DeserializerFeedback;
END_VAR
VAR
	timeAsString : T_MAXSTRING;
	error : I_Error;
END_VAR
IF NOT jsonParser.IsString(root) THEN
	error := errorFactory.CreateIncorrectTypeError('TOD');
	Feedback.LogError(error);
	RETURN;
END_IF

timeAsString := jsonParser.GetString(root);
Destination := STRING_TO_TOD(timeAsString);

TryGetTod := TRUE;
END_METHOD

METHOD TryGetUdint : BOOL
VAR_INPUT
	Destination : REFERENCE TO UDINT;
	Feedback : I_DeserializerFeedback;
END_VAR
VAR
	value : UDINT;
	error : I_Error;
END_VAR
IF NOT TryReadNumber(root, value) THEN
	error := errorFactory.CreateIncorrectTypeError('UDINT');
	Feedback.LogError(error);
	RETURN;
END_IF

Destination := value;
TryGetUdint := TRUE;
END_METHOD

METHOD TryGetUint : BOOL
VAR_INPUT
	Destination : REFERENCE TO UINT;
	Feedback : I_DeserializerFeedback;
END_VAR
VAR
	value : UINT;
	error : I_Error;
END_VAR
IF NOT TryReadNumber(root, value) THEN
	error := errorFactory.CreateIncorrectTypeError('UINT');
	Feedback.LogError(error);
	RETURN;
END_IF

Destination := value;
TryGetUint := TRUE;
END_METHOD

METHOD TryGetUlint : BOOL
VAR_INPUT
	Destination : REFERENCE TO ULINT;
	Feedback : I_DeserializerFeedback;
END_VAR
VAR
	value : ULINT;
	error : I_Error;
END_VAR
IF NOT TryReadNumber(root, value) THEN
	error := errorFactory.CreateIncorrectTypeError('ULINT');
	Feedback.LogError(error);
	RETURN;
END_IF

Destination := value;
TryGetUlint := TRUE;
END_METHOD

METHOD TryGetUsint : BOOL
VAR_INPUT
	Destination : REFERENCE TO USINT;
	Feedback : I_DeserializerFeedback;
END_VAR
VAR
	value : USINT;
	error : I_Error;
END_VAR
IF NOT TryReadNumber(root, value) THEN
	error := errorFactory.CreateIncorrectTypeError('USINT');
	Feedback.LogError(error);
	RETURN;
END_IF

Destination := value;
TryGetUsint := TRUE;
END_METHOD

METHOD TryGetWord : BOOL
VAR_INPUT
	Destination : REFERENCE TO WORD;
	Feedback : I_DeserializerFeedback;
END_VAR
VAR
	value : WORD;
	error : I_Error;
END_VAR
IF NOT TryReadNumber(root, value) THEN
	error := errorFactory.CreateIncorrectTypeError('WORD');
	Feedback.LogError(error);
	RETURN;
END_IF

Destination := value;
TryGetWord := TRUE;
END_METHOD

END_FUNCTION_BLOCK

// mobject-json/_Internal/JsonDeserializerForwardEnumerator/JsonDeserializerObjectForwardEnumerator
{attribute 'linkalways'} 
{attribute 'no_explicit_call' := 'This FB is a CLASS and must be accessed using methods or properties'}
{attribute 'enable_dynamic_creation'}
FUNCTION_BLOCK JsonDeserializerObjectForwardEnumerator EXTENDS Disposable IMPLEMENTS I_DeserializerObjectForwardEnumerator, I_EventHandler
VAR
	parent : I_JsonDeserializer;
	jsonParser : REFERENCE TO JsonDomParser;
	root : SJsonValue;
	garbageCollector : I_DeserializerGarbageCollector;
	nullNode : I_Deserializer;
	moveNextCalled : BOOL := FALSE;
	invalid : BOOL := FALSE; 
	nextMemberPosition : SJsonValue;
	memberBeginPosition : SJsonValue;
	memberEndPosition : SJsonValue;
	currentDeserializer : I_Deserializer;
	currentKey : T_MAXSTRING;
END_VAR

METHOD FB_init : BOOL
VAR_INPUT
	bInitRetains : BOOL; // if TRUE, the retain variables are initialized (warm start / cold start)
	bInCopyCode : BOOL;  // if TRUE, the instance afterwards gets moved into the copy code (online change)
	ParentJsonDeserializer : I_JsonDeserializer;
	ParentJsonDomParser : REFERENCE TO JsonDomParser;
	NodeRoot : SJsonValue;
	ParentGarbageCollector : I_DeserializerGarbageCollector;
	ParentNullDeserializer : I_Deserializer;
END_VAR
THIS^.parent := ParentJsonDeserializer;
THIS^.jsonParser REF= ParentJsonDomParser;
THIS^.root := NodeRoot;
THIS^.garbageCollector := ParentGarbageCollector;
THIS^.nullNode := ParentNullDeserializer;

Initialize();

Parent.OnEvent('OnChanged',THIS^);
Parent.OnEvent('OnDisposed',THIS^);
END_METHOD

METHOD FB_exit : BOOL
VAR_INPUT
	bInCopyCode : BOOL; // if TRUE, the exit method is called for exiting an instance that is copied afterwards (online change).
END_VAR
IF bInCopyCode THEN
	RETURN;
END_IF

IF parent = 0 THEN
	RETURN;
END_IF

parent.OffEvent('OnChanged',THIS^);
parent.OffEvent('OnDisposed',THIS^);
END_METHOD

METHOD PROTECTED CreateDeserializer : I_Deserializer
VAR_INPUT
	DeserializerRoot : SJsonValue;
END_VAR
VAR 
	pNode : POINTER TO JsonDeserializerNode;
END_VAR
pNode := __NEW(JsonDeserializerNode(
	ParentJsonDeserializer := parent,
	ParentJsonDomParser := jsonParser, 
	NodeRoot := DeserializerRoot, 
	ParentGarbageCollector := garbageCollector, 
	ParentNullDeserializer := nullNode
));

CreateDeserializer := pNode^;
END_METHOD

METHOD PROTECTED Initialize
VAR_INPUT
END_VAR
IF NOT jsonParser.IsObject(root) THEN
	invalid := TRUE;
	RETURN;
END_IF

memberBeginPosition := jsonParser.MemberBegin(root);
memberEndPosition := jsonParser.MemberEnd(root);

IF memberBeginPosition = 0 THEN
	invalid := TRUE;
	RETURN;
END_IF

IF memberEndPosition = 0 THEN
	invalid := TRUE;
	RETURN;
END_IF
END_METHOD

METHOD PROTECTED UpdateCurrentDeserializer
VAR_INPUT
	UpdatedRoot : SJsonValue;
END_VAR
VAR
	rootOfValue : SJsonValue;
END_VAR
IF currentDeserializer <> 0 THEN
	currentDeserializer.Dispose();
	currentDeserializer := 0;
END_IF

IF invalid THEN
	RETURN;
END_IF

rootOfValue := jsonParser.GetMemberValue(UpdatedRoot);
currentKey := jsonParser.GetMemberName(UpdatedRoot);

IF rootOfValue = 0 THEN
	RETURN;
END_IF

currentDeserializer := CreateDeserializer(rootOfValue);
END_METHOD

PROPERTY PUBLIC Current : I_Deserializer
GET
IF NOT IsValid THEN
	Current := nullNode;
	RETURN;
END_IF

IF currentDeserializer = 0 THEN
	Current := nullNode;
	RETURN;
END_IF

Current := currentDeserializer;
END_GET
END_PROPERTY

METHOD PUBLIC HandleEvent
VAR_INPUT
	Event : I_Event;
END_VAR
VAR
	changedEvent : I_JsonDeserializerChangedEvent;
	disposedEvent : I_JsonDeserializerDisposedEvent;
END_VAR
IF __QUERYINTERFACE(Event, changedEvent) THEN
	invalid := TRUE;
ELSIF __QUERYINTERFACE(Event, disposedEvent) THEN
	parent := 0;
	Dispose();
END_IF
END_METHOD

PROPERTY PUBLIC IsValid : BOOL
GET
PUBLIC
IF invalid THEN
	RETURN;
END_IF

IF parent = 0 THEN
	RETURN;
END_IF

IsValid := TRUE;
END_GET
END_PROPERTY

PROPERTY Key : T_MAXSTRING
GET
Key := currentKey;
END_GET
END_PROPERTY

METHOD PUBLIC MoveNext : BOOL
IF invalid THEN
    RETURN;
END_IF

// Handle the initial move
IF NOT moveNextCalled THEN
    moveNextCalled := TRUE;
    UpdateCurrentDeserializer(memberBeginPosition);
	nextMemberPosition := jsonParser.NextMember(memberBeginPosition);
	MoveNext := TRUE;
    RETURN;
END_IF

// Handle subsequent moves
IF nextMemberPosition <> memberEndPosition THEN	
	UpdateCurrentDeserializer(nextMemberPosition);
	nextMemberPosition := jsonParser.NextMember(nextMemberPosition);
	MoveNext := TRUE;
END_IF
END_METHOD

END_FUNCTION_BLOCK

// mobject-json/JsonDeserializer/JsonDeserializer
{attribute 'linkalways'} 
{attribute 'no_explicit_call' := 'This FB is a CLASS and must be accessed using methods or properties'}
{attribute 'enable_dynamic_creation'}
FUNCTION_BLOCK JsonDeserializer EXTENDS Disposable IMPLEMENTS I_JsonDeserializer
VAR
	jsonParser : JsonDomParser;
	root : SJsonValue;
	garbageCollector : DeserializerGarbageCollector;
	nullNode : JsonDeserializerNullNode(THIS^);
	rootNode : I_Deserializer := nullNode;
	eventEmitter : EventEmitter;
END_VAR

METHOD FB_exit : BOOL
VAR_INPUT
	bInCopyCode : BOOL; // if TRUE, the exit method is called for exiting an instance that is copied afterwards (online change).
END_VAR
IF bInCopyCode THEN
	RETURN;
END_IF

Reset();
EmitDisposedEvent();
END_METHOD

METHOD PROTECTED CreateDeserializer : I_Deserializer
VAR_INPUT
	DeserializerRoot : SJsonValue;
END_VAR
VAR 
	pNode : POINTER TO JsonDeserializerNode;
END_VAR
pNode := __NEW(JsonDeserializerNode(
	ParentJsonDeserializer := THIS^,
	ParentJsonDomParser := jsonParser, 
	NodeRoot := DeserializerRoot, 
	ParentGarbageCollector := garbageCollector, 
	ParentNullDeserializer := nullNode)
);

CreateDeserializer := pNode^;
END_METHOD

METHOD PRIVATE EmitChangedEvent
VAR
	pJsonDeserializerChangedEvent : POINTER TO JsonDeserializerChangedEvent;
END_VAR
pJsonDeserializerChangedEvent := __NEW(JsonDeserializerChangedEvent(Target := THIS^));
eventEmitter.Emit('OnChanged', pJsonDeserializerChangedEvent^);
pJsonDeserializerChangedEvent^.Dispose();
END_METHOD

METHOD PRIVATE EmitDisposedEvent
VAR
	pJsonDeserializerDisposedEvent : POINTER TO JsonDeserializerDisposedEvent;
END_VAR
pJsonDeserializerDisposedEvent := __NEW(JsonDeserializerDisposedEvent(Target := THIS^));
eventEmitter.Emit('OnDisposed', pJsonDeserializerDisposedEvent^);
pJsonDeserializerDisposedEvent^.Dispose();
END_METHOD

METHOD PUBLIC Clone : I_Deserializer
VAR
	pClone : POINTER TO JsonDeserializer;
	jsonSize : UDINT;
	pJsonString : POINTER TO STRING;
END_VAR
pClone := __NEW(JsonDeserializer);
Clone := pClone^;

jsonSize := jsonParser.GetDocumentLength();

IF jsonSize = 0 THEN
	// no further cloning to do. 
	RETURN;
END_IF

pJsonString := __NEW(BYTE, jsonSize);

IF jsonParser.CopyDocument(pJsonString^, jsonSize) = 0 THEN
	__DELETE(pJsonString);
	RETURN;
END_IF

pClone^.TryLoad(pJsonString^);
__DELETE(pJsonString);
END_METHOD

METHOD GetArray : I_Deserializer
VAR_INPUT
END_VAR
GetArray := rootNode.GetArray();
END_METHOD

METHOD GetArrayEnumerator : I_DeserializerArrayForwardEnumerator
VAR_INPUT
END_VAR
GetArrayEnumerator := rootNode.GetArrayEnumerator();
END_METHOD

METHOD GetElementByIndex : I_Deserializer
VAR_INPUT
	Index : UDINT;
END_VAR
GetElementByIndex := rootNode.GetElementByIndex(Index);
END_METHOD

METHOD GetKeyArray : I_Deserializer
VAR_INPUT
	Key : T_MAXSTRING;
END_VAR
GetKeyArray := rootNode.GetKeyArray(Key);
END_METHOD

METHOD GetKeyObject : I_Deserializer
VAR_INPUT
	Key : T_MAXSTRING;
END_VAR
GetKeyObject := rootNode.GetKeyObject(Key);
END_METHOD

METHOD GetObject : I_Deserializer
VAR_INPUT
END_VAR
GetObject := rootNode.GetObject();
END_METHOD

METHOD GetObjectEnumerator : I_DeserializerObjectForwardEnumerator
VAR_INPUT
END_VAR
GetObjectEnumerator := rootNode.GetObjectEnumerator();
END_METHOD

METHOD PUBLIC OffEvent
VAR_INPUT
	EventName : T_MaxString;
	EventHandler : I_EventHandler;
END_VAR
eventEmitter.OffEvent(EventName, EventHandler);
END_METHOD

METHOD PUBLIC OnceEvent
VAR_INPUT
	EventName : T_MaxString;
	EventHandler : I_EventHandler;
END_VAR
eventEmitter.OnceEvent(EventName, EventHandler);
END_METHOD

METHOD PUBLIC OnEvent
VAR_INPUT
	EventName : T_MaxString;
	EventHandler : I_EventHandler;
END_VAR
eventEmitter.OnEvent(EventName, EventHandler);
END_METHOD

METHOD PUBLIC Reset
VAR_INPUT
END_VAR
jsonParser.NewDocument();
garbageCollector.Execute();
root := 0;
rootNode := nullNode;
EmitChangedEvent();
END_METHOD

METHOD TryDeserializeKeyToObject : BOOL
VAR_INPUT
	Key : T_MAXSTRING;
	Object : I_Deserializable;
	Feedback : I_DeserializerFeedback;
END_VAR
TryDeserializeKeyToObject := rootNode.TryDeserializeKeyToObject(Key,Object, Feedback);
END_METHOD

METHOD TryDeserializeToObject : BOOL
VAR_INPUT
	Object : I_Deserializable;
	Feedback : I_DeserializerFeedback;
END_VAR
TryDeserializeToObject := rootNode.TryDeserializeToObject(Object, Feedback);
END_METHOD

METHOD TryGetBase64 : BOOL
VAR_INPUT
	pBytes : POINTER TO BYTE;
	nBytes : DINT;
	Feedback : I_DeserializerFeedback;
END_VAR
TryGetBase64 := rootNode.TryGetBase64(pBytes, nBytes, Feedback);
END_METHOD

METHOD TryGetBool : BOOL
VAR_INPUT
	Destination : REFERENCE TO BOOL;
	Feedback : I_DeserializerFeedback;
END_VAR
TryGetBool := rootNode.TryGetBool(Destination, Feedback);
END_METHOD

METHOD TryGetByte : BOOL
VAR_INPUT
	Destination : REFERENCE TO BYTE;
	Feedback : I_DeserializerFeedback;
END_VAR
TryGetByte := rootNode.TryGetByte(Destination, Feedback);
END_METHOD

METHOD TryGetDateTime : BOOL
VAR_INPUT
	Destination : REFERENCE TO DATE_AND_TIME;
	Feedback : I_DeserializerFeedback;
END_VAR
TryGetDateTime := rootNode.TryGetDateTime(Destination, Feedback);
END_METHOD

METHOD TryGetDcTime : BOOL
VAR_INPUT
	Destination : REFERENCE TO DCTIME;
	Feedback : I_DeserializerFeedback;
END_VAR
TryGetDcTime := rootNode.TryGetDcTime(Destination, Feedback);
END_METHOD

METHOD TryGetDint : BOOL
VAR_INPUT
	Destination : REFERENCE TO DINT;
	Feedback : I_DeserializerFeedback;
END_VAR
TryGetDint := rootNode.TryGetDint(Destination, Feedback);
END_METHOD

METHOD TryGetDword : BOOL
VAR_INPUT
	Destination : REFERENCE TO DWORD;
	Feedback : I_DeserializerFeedback;
END_VAR
TryGetDword := rootNode.TryGetDword(Destination, Feedback);
END_METHOD

METHOD TryGetElementByIndex : BOOL
VAR_INPUT
	Index : UDINT;
	Destination : REFERENCE TO I_Deserializer;
	Feedback : I_DeserializerFeedback;
END_VAR
TryGetElementByIndex := rootNode.TryGetElementByIndex(Index, Destination, Feedback);
END_METHOD

METHOD TryGetFileTime : BOOL
VAR_INPUT
	Destination : REFERENCE TO FILETIME;
	Feedback : I_DeserializerFeedback;
END_VAR
TryGetFileTime := rootNode.TryGetFileTime(Destination, Feedback);
END_METHOD

METHOD TryGetHexAsBytes : BOOL
VAR_INPUT
	pBytes : POINTER TO BYTE;
	nBytes : DINT;
	Feedback : I_DeserializerFeedback;
END_VAR
TryGetHexAsBytes := rootNode.TryGetHexAsBytes(pBytes, nBytes, Feedback);
END_METHOD

METHOD TryGetInt : BOOL
VAR_INPUT
	Destination : REFERENCE TO INT;
	Feedback : I_DeserializerFeedback;
END_VAR
TryGetInt := rootNode.TryGetInt(Destination, Feedback);
END_METHOD

METHOD TryGetKeyBase64 : BOOL
VAR_INPUT
	Key : T_MAXSTRING;
	pBytes : POINTER TO BYTE;
	nBytes : DINT;
	Feedback : I_DeserializerFeedback;
END_VAR
TryGetKeyBase64 := rootNode.TryGetKeyBase64(Key, pBytes, nBytes, Feedback);
END_METHOD

METHOD TryGetKeyBool : BOOL
VAR_INPUT
	Key : T_MAXSTRING;
	Destination : REFERENCE TO BOOL;
	Feedback : I_DeserializerFeedback;
END_VAR
TryGetKeyBool := rootNode.TryGetKeyBool(Key, Destination, Feedback);
END_METHOD

METHOD TryGetKeyByte : BOOL
VAR_INPUT
	Key : T_MAXSTRING;
	Destination : REFERENCE TO BYTE;
	Feedback : I_DeserializerFeedback;
END_VAR
TryGetKeyByte := rootNode.TryGetKeyByte(Key, Destination, Feedback);
END_METHOD

METHOD TryGetKeyDateTime : BOOL
VAR_INPUT
	Key : T_MAXSTRING;
	Destination : REFERENCE TO DATE_AND_TIME;
	Feedback : I_DeserializerFeedback;
END_VAR
TryGetKeyDateTime := rootNode.TryGetKeyDateTime(Key, Destination, Feedback);
END_METHOD

METHOD TryGetKeyDcTime : BOOL
VAR_INPUT
	Key : T_MAXSTRING;
	Destination : REFERENCE TO DCTIME;
	Feedback : I_DeserializerFeedback;
END_VAR
TryGetKeyDcTime := rootNode.TryGetKeyDcTime(Key, Destination, Feedback);
END_METHOD

METHOD TryGetKeyDint : BOOL
VAR_INPUT
	Key : T_MAXSTRING;
	Destination : REFERENCE TO DINT;
	Feedback : I_DeserializerFeedback;
END_VAR
TryGetKeyDint := rootNode.TryGetKeyDint(Key, Destination, Feedback);
END_METHOD

METHOD TryGetKeyDword : BOOL
VAR_INPUT
	Key : T_MAXSTRING;
	Destination : REFERENCE TO DWORD;
	Feedback : I_DeserializerFeedback;
END_VAR
TryGetKeyDword := rootNode.TryGetKeyDword(Key, Destination, Feedback);
END_METHOD

METHOD TryGetKeyFileTime : BOOL
VAR_INPUT
	Key : T_MAXSTRING;
	Destination : REFERENCE TO FILETIME;
	Feedback : I_DeserializerFeedback;
END_VAR
TryGetKeyFileTime := rootNode.TryGetKeyFileTime(Key, Destination, Feedback);
END_METHOD

METHOD TryGetKeyHexAsBytes : BOOL
VAR_INPUT
	Key : T_MAXSTRING;
	pBytes : POINTER TO BYTE;
	nBytes : DINT;
	Feedback : I_DeserializerFeedback;
END_VAR
TryGetKeyHexAsBytes := rootNode.TryGetKeyHexAsBytes(Key, pBytes, nBytes, Feedback);
END_METHOD

METHOD TryGetKeyInt : BOOL
VAR_INPUT
	Key : T_MAXSTRING;
	Destination : REFERENCE TO INT;
	Feedback : I_DeserializerFeedback;
END_VAR
TryGetKeyInt := rootNode.TryGetKeyInt(Key, Destination, Feedback);
END_METHOD

METHOD TryGetKeyLint : BOOL
VAR_INPUT
	Key : T_MAXSTRING;
	Destination : REFERENCE TO LINT;
	Feedback : I_DeserializerFeedback;
END_VAR
TryGetKeyLint := rootNode.TryGetKeyLint(Key, Destination, Feedback);
END_METHOD

METHOD TryGetKeyLreal : BOOL
VAR_INPUT
	Key : T_MAXSTRING;
	Destination : REFERENCE TO LREAL;
	Feedback : I_DeserializerFeedback;
END_VAR
TryGetKeyLreal := rootNode.TryGetKeyLreal(Key, Destination, Feedback);
END_METHOD

METHOD TryGetKeyLtime : BOOL
VAR_INPUT
	Key : T_MAXSTRING;
	Destination : REFERENCE TO LTIME;
	Feedback : I_DeserializerFeedback;
END_VAR
TryGetKeyLtime := rootNode.TryGetKeyLtime(Key, Destination, Feedback);
END_METHOD

METHOD TryGetKeyLword : BOOL
VAR_INPUT
	Key : T_MAXSTRING;
	Destination : REFERENCE TO LWORD;
	Feedback : I_DeserializerFeedback;
END_VAR
TryGetKeyLword := rootNode.TryGetKeyLword(Key, Destination, Feedback);
END_METHOD

METHOD TryGetKeyReal : BOOL
VAR_INPUT
	Key : T_MAXSTRING;
	Destination : REFERENCE TO REAL;
	Feedback : I_DeserializerFeedback;
END_VAR
TryGetKeyReal := rootNode.TryGetKeyReal(Key, Destination, Feedback);
END_METHOD

METHOD TryGetKeySint : BOOL
VAR_INPUT
	Key : T_MAXSTRING;
	Destination : REFERENCE TO SINT;
	Feedback : I_DeserializerFeedback;
END_VAR
TryGetKeySint := rootNode.TryGetKeySint(Key, Destination, Feedback);
END_METHOD

METHOD TryGetKeyString : BOOL
VAR_INPUT
	Key : T_MAXSTRING;
	Destination : REFERENCE TO T_MAXSTRING;
	Feedback : I_DeserializerFeedback;
END_VAR
TryGetKeyString := rootNode.TryGetKeyString(Key, Destination, Feedback);
END_METHOD

METHOD TryGetKeyStringEx : BOOL
VAR_INPUT
	Key : T_MAXSTRING;
	DestinationAddress : POINTER TO STRING;
	DestinationSize : UDINT;
	Feedback : I_DeserializerFeedback;
END_VAR
TryGetKeyStringEx := rootNode.TryGetKeyStringEx(Key, DestinationAddress, DestinationSize, Feedback);
END_METHOD

METHOD TryGetKeyTime : BOOL
VAR_INPUT
	Key : T_MAXSTRING;
	Destination : REFERENCE TO TIME;
	Feedback : I_DeserializerFeedback;
END_VAR
TryGetKeyTime := rootNode.TryGetKeyTime(Key, Destination, Feedback);
END_METHOD

METHOD TryGetKeyTod : BOOL
VAR_INPUT
	Key : T_MAXSTRING;
	Destination : REFERENCE TO TOD;
	Feedback : I_DeserializerFeedback;
END_VAR
TryGetKeyTod := rootNode.TryGetKeyTod(Key, Destination, Feedback);
END_METHOD

METHOD TryGetKeyUdint : BOOL
VAR_INPUT
	Key : T_MAXSTRING;
	Destination : REFERENCE TO UDINT;
	Feedback : I_DeserializerFeedback;
END_VAR
TryGetKeyUdint := rootNode.TryGetKeyUdint(Key, Destination, Feedback);
END_METHOD

METHOD TryGetKeyUint : BOOL
VAR_INPUT
	Key : T_MAXSTRING;
	Destination : REFERENCE TO UINT;
	Feedback : I_DeserializerFeedback;
END_VAR
TryGetKeyUint := rootNode.TryGetKeyUint(Key, Destination, Feedback);
END_METHOD

METHOD TryGetKeyUlint : BOOL
VAR_INPUT
	Key : T_MAXSTRING;
	Destination : REFERENCE TO ULINT;
	Feedback : I_DeserializerFeedback;
END_VAR
TryGetKeyUlint := rootNode.TryGetKeyUlint(Key, Destination, Feedback);
END_METHOD

METHOD TryGetKeyUsint : BOOL
VAR_INPUT
	Key : T_MAXSTRING;
	Destination : REFERENCE TO USINT;
	Feedback : I_DeserializerFeedback;
END_VAR
TryGetKeyUsint := rootNode.TryGetKeyUsint(Key, Destination, Feedback);
END_METHOD

METHOD TryGetKeyWord : BOOL
VAR_INPUT
	Key : T_MAXSTRING;
	Destination : REFERENCE TO WORD;
	Feedback : I_DeserializerFeedback;
END_VAR
TryGetKeyWord := rootNode.TryGetKeyWord(Key, Destination, Feedback);
END_METHOD

METHOD TryGetLint : BOOL
VAR_INPUT
	Destination : REFERENCE TO LINT;
	Feedback : I_DeserializerFeedback;
END_VAR
TryGetLint := rootNode.TryGetLint(Destination, Feedback);
END_METHOD

METHOD TryGetLreal : BOOL
VAR_INPUT
	Destination : REFERENCE TO LREAL;
	Feedback : I_DeserializerFeedback;
END_VAR
TryGetLreal := rootNode.TryGetLreal(Destination, Feedback);
END_METHOD

